                uiBothStep := 1000;

            1000:
                IF Get THEN // Get box job

                    CASE Address_A OF
                        1:
                            DAS_CoreSys.MachineControl.fballocatearea
                                .M_StartStoragePulloutAction(CommandType := E_PullOutConveyorCommandType.SlideB_FeedIn_Ext,
                                                             CV_BackwardTIme := T#0S,
                                                             CV_ForwardTime := T#0S);
                        2:
                            DAS_CoreSys.MachineControl.fballocatearea
                                .M_StartStoragePulloutAction(CommandType := E_PullOutConveyorCommandType.SlideA_FeedIn_Ext,
                                                             CV_BackwardTIme := T#0S,
                                                             CV_ForwardTime := T#0S);
                    END_CASE

                ELSE
                    CASE Address_A OF
                        1:
                            DAS_CoreSys.MachineControl.fballocatearea
                                .M_StartStoragePulloutAction(CommandType := E_PullOutConveyorCommandType.SlideB_FeedOut_Ext,
                                                             CV_BackwardTIme := T#2S,
                                                             CV_ForwardTime := T#0S);

                        2:
                            DAS_CoreSys.MachineControl.fballocatearea
                                .M_StartStoragePulloutAction(CommandType := E_PullOutConveyorCommandType.SlideA_FeedOut_Ext,
                                                             CV_BackwardTIme := T#2S,
                                                             CV_ForwardTime := T#0S);
                    END_CASE

                END_IF

                uiBothStep := 1100;
            1100:
                IF DAS_CoreSys.MachineControl.fballocatearea.fbPulloutCv.Done THEN
                    DAS_CoreSys.MachineControl.fballocatearea.M_StopStoragePulloutAction();
                    BoxReady_1st := TRUE;
                    uiBothStep := 2000;
                END_IF

                IF DAS_CoreSys.MachineControl.fballocatearea.fbPulloutCv.Error THEN
                    DAS_CoreSys.MachineControl.fballocatearea.M_StopStoragePulloutAction();
                    uiResumeStep := 30000;
                    uiBothStep := 1000;
                    _Abort := TRUE;
                    strStatus := 'Feed box timeout';
                END_IF

            2000:
                IF Robot._DI1.Notification THEN
                    uiBothStep := 3000;
                END_IF
            3000:

                IF Get THEN // Get box job

                    CASE Address_B OF
                        1:
                            DAS_CoreSys.MachineControl.fballocatearea
                                .M_StartStoragePulloutAction(CommandType := E_PullOutConveyorCommandType.SlideB_FeedIn_Ext,
                                                             CV_BackwardTIme := T#0S,
                                                             CV_ForwardTime := T#0S);
                        2:
                            DAS_CoreSys.MachineControl.fballocatearea
                                .M_StartStoragePulloutAction(CommandType := E_PullOutConveyorCommandType.SlideA_FeedIn_Ext,
                                                             CV_BackwardTIme := T#0S,
                                                             CV_ForwardTime := T#0S);
                    END_CASE

                ELSE
                    CASE Address_B OF
                        1:
                            DAS_CoreSys.MachineControl.fballocatearea
                                .M_StartStoragePulloutAction(CommandType := E_PullOutConveyorCommandType.SlideB_FeedOut_Ext,
                                                             CV_BackwardTIme := T#2S,
                                                             CV_ForwardTime := T#0S);

                        2:
                            DAS_CoreSys.MachineControl.fballocatearea
                                .M_StartStoragePulloutAction(CommandType := E_PullOutConveyorCommandType.SlideA_FeedOut_Ext,
                                                             CV_BackwardTIme := T#2S,
                                                             CV_ForwardTime := T#0S);
                    END_CASE
                END_IF

                uiBothStep := 3100;
            3100:
                IF DAS_CoreSys.MachineControl.fballocatearea.fbPulloutCv.Done THEN
                    DAS_CoreSys.MachineControl.fballocatearea.M_StopStoragePulloutAction();
                    BoxReady_2nd := TRUE;
                    uiBothStep := 9999;
                END_IF

                IF DAS_CoreSys.MachineControl.fballocatearea.fbPulloutCv.Error THEN
                    DAS_CoreSys.MachineControl.fballocatearea.M_StopStoragePulloutAction();
                    uiResumeStep := 30000;
                    uiBothStep := 3000;
                    _Abort := TRUE;
                    strStatus := 'Feed box timeout';
                END_IF
            9999: //Wait		
        // wait reset
        END_CASE

        // Robot Abs move
        Robot.M_StartRobotAbsMove(GetBox := Get,
                                  UseClampA := UseA,
                                  UseClampB := UseB,
                                  Area := Area,
                                  ClampA_Address := Address_A,
                                  ClampB_Address := Address_B,
                                  BoxReady_1 := BoxReady_1st,
                                  BoxReady_2 := BoxReady_2nd);

        IF Robot._DI1.Done THEN
            tonTimeOut.IN := FALSE;
            uiExecutingStep := 30080;
        END_IF

        tonTimeOut.IN := TRUE;

        IF tonTimeOut.Q = TRUE THEN
            tonTimeOut.IN := FALSE;
            strStatus := 'Reset Robot timeout';
            _Error := TRUE;
        END_IF
    30080: // Check robot command is clear

        Robot.M_ResetRobotAbsMove(UseA, UseB);
        DAS_CoreSys.MachineControl.fballocatearea.M_StopStoragePulloutAction();

        IF NOT Robot._DI1.Done THEN
            tonTimeOut.IN := FALSE;
            uiExecutingStep := 99000; // 
        END_IF

        tonTimeOut.IN := TRUE;

        IF tonTimeOut.Q = TRUE THEN
            strStatus := 'Stop Robot timeout';
            _Error := TRUE;
        END_IF

    99000: // process done
        DAS_CoreSys.MachineControl.fballocatearea.M_ReleasePulloutAccess(ControlAccess := E_RoundBeltControlAccess.FanucRobot);
        Status := 'Process completed';
        _Executed := TRUE;
END_CASE

IF _Executed THEN
    eState := STATE_DONE;
ELSIF _Error THEN
    //	FUN_UniqueErrorCodeGenerator(iErrorID := ErrorID,UinqueErrorCode=>_UniqueErrorCode);
    eState := STATE_ERROR;
ELSIF NOT Execute THEN
    eState := STATE_RESETTING;
END_IF

IF _Abort OR Abort THEN
    //	FUN_UniqueErrorCodeGenerator(iErrorID := ErrorID,UinqueErrorCode=>_UniqueErrorCode);
    eSTATE := STATE_ABORTING;
END_IF
END_METHOD

METHOD  M_STATE_RESETTING
VAR_INPUT
END_VAR
Error := FALSE;
Done := FALSE;
Busy := FALSE;

CASE uiResettingStep OF

    0:
        tonTimeOut.IN := FALSE;
        Robot.M_ResetAllCommand();
        Robot.M_ResetRobotAbsMove(TRUE, TRUE);
        uiResettingStep := 100;
        DAS_CoreSys.MachineControl.fbStorageArea.M_ResetSlides_FeedOut();
    100:

        // DAS_CoreSys.MachineControl.fbStorageArea.M_InactivePulloutConveyorInternCtrl();
        DAS_CoreSys.MachineControl.fbAllocateArea.M_ReleasePulloutAccess(ControlAccess := E_RoundBeltControlAccess.FanucRobot);
        DAS_CoreSys.MachineControl.fbAllocateArea.M_StopStoragePulloutAction();
        uiResettingStep := 9999;
    9999:
        _ResetCompleted := TRUE;
END_CASE

IF _ResetCompleted THEN
    eSTATE := STATE_DORMANT;
END_IF
END_METHOD

END_FUNCTION_BLOCK

// ---- Library/20_MachineUnits/21_StorageArea/Service/FB_RobotRegionMove_RoundBelt.TcPOU
FUNCTION_BLOCK FB_RobotRegionMove_RoundBelt EXTENDS FB_ObjectBase_V2 IMPLEMENTS IBasicElement
VAR_INPUT
    Robot     					: REFERENCE TO FB_FanucRobot_Basic;
	RoundBelt					: REFERENCE TO FB_RoundBeltService;	
   // Command   : ST_WareHouseWithRobotMove_Command;
    Info	  : ST_RobotRegionMove_Info;
	Input : ST_InputTable;
	Stop	  : BOOL;
END_VAR
VAR_OUTPUT
  // Status : ST_WareHouseWithRobotMove_Status;
END_VAR
VAR
	_Abort		: BOOL;
	strStatus	: STRING;
	uiResumeStep : UINT;
	
	Area	: E_RobotArea :=E_RobotArea.RoundBelt;
	UseA 	: BOOL;
	UseB	: BOOL;
	
	Get 	:BOOL;
	tonTimeOut	:TON;
	tonCheckRoundBeltDelay	:TON;
	_UniqueErrorCode :STRING;
	PreviousStrStatus : STRING;
	PreviousErrorCode : STRING;
END_VAR

SUPER^.A10_StateControl();
A00_BasicUnits();

ACTION A00_BasicUnits:
tonTimeOut(PT:=T#60S);
tonCheckRoundBeltDelay(PT:=T#2S);
ErrorID:=2220;
END_ACTION

METHOD M_CheckCommand : BOOL // True : Command is useful
VAR_INPUT
END_VAR
VAR
	
END_VAR
// Check command paremeter is correct
	
THIS^.Get :=Info.Get;
UseA := Info.UseA;
UseB := Info.UseB;
	//Normal command : RoundBelt
		IF Info.UseA AND (Info.A_Position<1 OR  Info.A_Position>3) THEN
			strStatus:='Wrong command ,Position A Not allowed';
			M_CheckCommand:=FALSE;
			RETURN;			
		END_IF
		
	
	//Normal command : RoundBelt
		IF Info.UseB AND(Info.B_Position<1 OR  Info.B_Position>3) THEN
			strStatus:='Wrong command ,Position B Not allowed';
			M_CheckCommand:=FALSE;
			RETURN;				
		END_IF
		
	

M_CheckCommand:=TRUE;
END_METHOD

METHOD M_CheckUnitsNotBusy : BOOL
VAR_INPUT
END_VAR
M_CheckUnitsNotBusy := true;
END_METHOD

METHOD M_CheckUnitsReady : BOOL
VAR_INPUT
END_VAR
M_CheckUnitsReady := true;
END_METHOD

METHOD  M_STATE_ABORTED
VAR_INPUT
END_VAR
ERROR :=TRUE;
Busy    := FALSE;
Aborted := TRUE;
Status := strStatus;
UniqueErrorCode:=_UniqueErrorCode;
IF NOT Execute THEN
	eSTATE:=STATE_RESETTING;
END_IF

IF Execute AND Reset THEN
	PreviousStrStatus := strStatus;
	PreviousErrorCode := _UniqueErrorCode;
	uiExecutingStep :=uiResumeStep;
	eSTATE:=STATE_EXECUTING;
END_IF
END_METHOD

METHOD  M_STATE_ABORTING
VAR_INPUT
END_VAR
CASE uiAbortingStep OF
	0 :
		uiAbortingStep:=9999;
		tonTimeOut.IN :=FALSE;
		_Abort :=FALSE;
		IF strStatus = PreviousStrStatus THEN
			_UniqueErrorCode :=PreviousErrorCode;
		END_IF
	9999:	_AbortCompleted:=TRUE;
END_CASE

IF _AbortCompleted THEN	
	eSTATE :=STATE_ABORTED;
END_IF
END_METHOD

METHOD  M_STATE_DONE
VAR_INPUT
END_VAR
Busy := FALSE;
Done := TRUE;
IF NOT Execute THEN
    eState := STATE_RESETTING;
END_IF
END_METHOD

METHOD  M_STATE_DORMANT
VAR_INPUT
END_VAR
// Clear FB output
Busy            := FALSE;
Done            := FALSE;
Aborted         := FALSE;
Error           := FALSE;
ErrorID         := 0;
Status          := '';
_ResetCompleted := FALSE;
_Error          := FALSE;
_Executed       := FALSE;

tonTimeOut.IN:=tonCheckRoundBeltDelay.IN:= FALSE;
strStatus :='No Error';
uiExecutingStep :=uiResettingStep :=uiResumeStep :=0;
PreviousStrStatus			 :='';
PreviousErrorCode			 :='';

// Wait Execute command
IF Execute THEN
    eState := STATE_EXECUTING;
END_IF
END_METHOD

METHOD  M_STATE_ERROR
VAR_INPUT
END_VAR
ERROR   :=TRUE;
Busy	:=FALSE;
Status := strStatus;
UniqueErrorCode:=_UniqueErrorCode;
IF NOT Execute THEN	
eSTATE:=STATE_RESETTING;
END_IF
END_METHOD

METHOD  M_STATE_EXECUTING
VAR_INPUT
END_VAR
VAR_INST
	BoxReady_1st : BOOL;
	BoxReady_2nd : BOOL;
    uiBothStep : UINT;
    uiSingleClampStep : UINT;	
	Address_A : INT;
	Address_B : INT;
	A1Used	 : BOOL;
	A2Used	 : BOOL;
END_VAR
VAR
	
	
END_VAR
//20250418 note: current behavior : wait round belt finish rotating then check if box is ready , everything ready then call Robot start move
//				 Todo : consider if better call robot start move to waiting position and check box at same moment , Albert 

// Set Busy active edit by johnson
Busy := TRUE;
IF THIS^.Stop THEN // Pending the timeout when Stop signal occur
	tonTimeout.IN :=FALSE;
END_IF
// Service Process
CASE uiExecutingStep OF
	0:
        // Clear variable      
        uiBothStep := 0;
		uiSingleClampStep :=0;
		BoxReady_1st := 0;
		BoxReady_2nd := 0;
		tonTimeOut.IN:=FALSE;
		tonCheckRoundBeltDelay.IN :=FALSE;
        // Check command
        IF M_CheckCommand() THEN
            uiExecutingStep := 10;
		ELSE
			_Error:=TRUE;
        END_IF
    10:
        // Start process, check units first
        IF M_CheckUnitsReady() THEN
            uiExecutingStep := 20;
        END_IF
    20:
        // CHeck units not busy state
        IF M_CheckUnitsNotBusy() THEN
            uiExecutingStep := 1000;
        END_IF
   
	1000:   
			// Read   coordinate
			 Area := THIS^.Area;
 			 Address_A := LREAL_TO_INT(Info.A_Position);
			 Address_B := LREAL_TO_INT(Info.B_Position);
			 uiExecutingStep := 1100; 		
			 
	1100:	
			// Check clamp userage	 
			IF UseA AND NOT UseB THEN
				//Only clampA
				uiExecutingStep := 10000;
			ELSIF NOT UseA AND UseB THEN
				//Only ClampB 
				uiExecutingStep := 20000;
			ELSIF UseA AND UseB THEN
				//Both Clamps
				uiExecutingStep := 30000;		
			END_IF
       
    10000: // Only ClampA 
        IF NOT Robot._DI1.Done THEN
			// Delay to make sure round belt is starting/finish rotating
			IF NOT RoundBelt.xBusy AND NOT RoundBelt.xError THEN
				tonCheckRoundBeltDelay.IN:=TRUE;
			ELSE
				tonCheckRoundBeltDelay.IN:=FALSE;	
			END_IF
		
		
		CASE uiSingleClampStep OF
		0:
			CASE Address_A OF						
						1: A1Used := TRUE;
						2: A2Used := TRUE;
			END_CASE
			
			IF tonCheckRoundBeltDelay.Q THEN
				IF Get THEN  // Picking job , check box is ready
					IF A1Used AND Input.bRoundBelt_ChangeZoneA2Detect_Sensor =FALSE	THEN
						_Error:=TRUE	;
						strStatus :='No Box on A1';
					END_IF				
					IF A2Used AND Input.bRoundBelt_ChangeZoneA3Detect_Sensor =FALSE	THEN
						_Error:=TRUE	;
						strStatus :='No Box on A2';
					END_IF	
				ELSE		//Place job , check no box 
					IF A1Used AND Input.bRoundBelt_ChangeZoneA2Detect_Sensor =TRUE	THEN
						_Error:=TRUE	;
						strStatus :='Box on A1';
					END_IF				
					IF A2Used AND Input.bRoundBelt_ChangeZoneA3Detect_Sensor =TRUE	THEN
						_Error:=TRUE	;
						strStatus :='Box on A2';
					END_IF				
				END_IF
				 uiSingleClampStep:=100;  
			END_IF
	  
		  100 :  
		  		IF get THEN
					BoxReady_1st := (A1Used AND Input.bRoundBelt_ChangeZoneA2Detect_Sensor) OR
		  						 (A2Used AND Input.bRoundBelt_ChangeZoneA3Detect_Sensor);
				ELSE
					BoxReady_1st := (A1Used AND NOT Input.bRoundBelt_ChangeZoneA2Detect_Sensor) OR
		  						 (A2Used AND NOT Input.bRoundBelt_ChangeZoneA3Detect_Sensor);
				END_IF		
				IF BoxReady_1st THEN
					uiSingleClampStep:=9999;  
				END_IF			 
								 
		  9999:// 
	
		END_CASE				          		 
				  // Robot Abs move
           		 Robot.M_StartRobotAbsMove(GetBox:=Get,
											UseClampA:=UseA,
											UseClampB:=UseB,
											Area:=Area,
											ClampA_Address:=Address_A,
											ClampB_Address:=Address_B,
											BoxReady_1:=BoxReady_1st,
											BoxReady_2:=BoxReady_2nd);				  
		
        ELSE
			tonTimeOut.IN:=FALSE;
            uiExecutingStep := 10080;
        END_IF
		tonTimeOut.IN:=TRUE;
		IF tonTimeOut.Q=TRUE THEN
			tonTimeOut.IN:=FALSE;
			strStatus :='Reset Robot timeout';
			_Error:=TRUE;
		END_IF	
    10080:
        Robot.M_ResetRobotAbsMove(UseA,UseB); // Clear command and go to place box
		tonTimeOut.IN:=TRUE;
        IF NOT Robot._DI1.Done THEN
			tonTimeOut.IN:=FALSE;
            uiExecutingStep := 99000; 
        END_IF
    	IF tonTimeOut.Q=TRUE THEN
			strStatus :='Reset Robot timeout';
			_Error:=TRUE;
		END_IF	
    
   20000: // Only ClampB
        IF NOT Robot._DI1.Done THEN
           IF NOT RoundBelt.xBusy AND NOT RoundBelt.xError THEN
				tonCheckRoundBeltDelay.IN:=TRUE;
			ELSE
				tonCheckRoundBeltDelay.IN:=FALSE;	
			END_IF
		
		
		CASE uiSingleClampStep OF
		0:
			CASE Address_B OF						
						1: A1Used := TRUE;
						2: A2Used := TRUE;
			END_CASE
			
			IF tonCheckRoundBeltDelay.Q THEN
				IF Get THEN  // Picking job , check box is ready
					IF A1Used AND Input.bRoundBelt_ChangeZoneA2Detect_Sensor =FALSE	THEN
						_Error:=TRUE	;
						strStatus :='No Box on A1';
					END_IF				
					IF A2Used AND Input.bRoundBelt_ChangeZoneA3Detect_Sensor =FALSE	THEN
						_Error:=TRUE	;
						strStatus :='No Box on A2';
					END_IF	
				ELSE		//Place job , check no box 
					IF A1Used AND Input.bRoundBelt_ChangeZoneA2Detect_Sensor =TRUE	THEN
						_Error:=TRUE	;
						strStatus :='Box on A1';
					END_IF				
					IF A2Used AND Input.bRoundBelt_ChangeZoneA3Detect_Sensor =TRUE	THEN
						_Error:=TRUE	;
						strStatus :='Box on A2';
					END_IF				
				END_IF
				 uiSingleClampStep:=100;  
			END_IF
	  
		  100 :  
		  		IF get THEN
					BoxReady_2nd := (A1Used AND Input.bRoundBelt_ChangeZoneA2Detect_Sensor) OR
		  						 (A2Used AND Input.bRoundBelt_ChangeZoneA3Detect_Sensor);
				ELSE
					BoxReady_2nd := (A1Used AND NOT Input.bRoundBelt_ChangeZoneA2Detect_Sensor) OR
		  						 (A2Used AND NOT Input.bRoundBelt_ChangeZoneA3Detect_Sensor);
				END_IF		
				IF BoxReady_2nd THEN
					uiSingleClampStep:=9999;  
				END_IF			 
								 
		  9999:// 
	
		END_CASE				          		 
					  // Robot Abs move
           		 Robot.M_StartRobotAbsMove( GetBox:=Get,
											UseClampA:=UseA,
											UseClampB:=UseB,
											Area:=Area,
											ClampA_Address:=Address_A,
											ClampB_Address:=Address_B,
											BoxReady_1:=BoxReady_1st,
											BoxReady_2:=BoxReady_2nd);		  
		
        ELSE
			tonTimeOut.IN:=FALSE;
            uiExecutingStep := 20080;
        END_IF	
		tonTimeOut.IN:=TRUE;
		IF tonTimeOut.Q=TRUE THEN
			tonTimeOut.IN:=FALSE;
			strStatus :='Reset Robot timeout';
			_Error:=TRUE;
		END_IF				          		 
			
       
		
    20080:
       Robot.M_ResetRobotAbsMove(UseA,UseB);; // Clear command 

        IF NOT Robot._DI1.Done THEN
            uiExecutingStep := 99000; 
        END_IF
		tonTimeOut.IN:=TRUE;
		IF tonTimeOut.Q=TRUE THEN
			strStatus :='Reset Robot timeout';
			_Error:=TRUE;
		END_IF	
    30000: // Both Clamps
        	
			IF NOT RoundBelt.xBusy AND NOT RoundBelt.xError THEN
				tonCheckRoundBeltDelay.IN:=TRUE;
			ELSE
				tonCheckRoundBeltDelay.IN:=FALSE;	
			END_IF
		
		  CASE uiBothStep OF
           		0://	
					BoxReady_1st := FALSE;
					BoxReady_2nd := FALSE;
					
					IF tonCheckRoundBeltDelay.Q THEN
						uiBothStep:=100;	
					END_IF
				100:
					IF Get THEN  // Picking job , check box is ready
						IF  Input.bRoundBelt_ChangeZoneA2Detect_Sensor =FALSE	THEN
							_Error:=TRUE	;
							strStatus :='No Box on A1';
						END_IF				
						IF  Input.bRoundBelt_ChangeZoneA3Detect_Sensor =FALSE	THEN
							_Error:=TRUE	;
							strStatus :='No Box on A2';
						END_IF	
					ELSE		//Place job , check no box 
						IF  Input.bRoundBelt_ChangeZoneA2Detect_Sensor =TRUE	THEN
							_Error:=TRUE	;
							strStatus :='Box on A1';
						END_IF				
						IF  Input.bRoundBelt_ChangeZoneA3Detect_Sensor =TRUE	THEN
							_Error:=TRUE	;
							strStatus :='Box on A2';
						END_IF				
					END_IF
					IF NOT _Error THEN
						uiBothStep:=1000;
					END_IF
				1000:	
						
						BoxReady_1st :=TRUE;
						uiBothStep:=2000;
					
						
				2000:					
						IF Robot._DI1.Notification THEN
							uiBothStep:=3000;
						END_IF
				3000:	
						 BoxReady_2nd :=TRUE;						 
					     uiBothStep:=9999;
				
				9999: //Wait		
        // wait reset
        END_CASE

       	  // Robot Abs move
           		 Robot.M_StartRobotAbsMove( GetBox:=Get,
											UseClampA:=UseA,
											UseClampB:=UseB,
											Area:=Area,
											ClampA_Address:=Address_A,
											ClampB_Address:=Address_B,
											BoxReady_1:=BoxReady_1st,
											BoxReady_2:=BoxReady_2nd);	
		
		
        IF Robot._DI1.Done THEN
			tonTimeOut.IN:=FALSE;
            uiExecutingStep := 30080;
        END_IF
		tonTimeOut.IN:=TRUE;
		IF tonTimeOut.Q=TRUE THEN
			tonTimeOut.IN:=FALSE;
			strStatus :='Reset Robot timeout';
			_Error:=TRUE;
		END_IF	
		
    30080: // Check robot command is clear
        
        Robot.M_ResetRobotAbsMove(UseA,UseB);

        IF NOT Robot._DI1.Done THEN
			tonTimeOut.IN:=FALSE;
            uiExecutingStep := 99000; // go to place step
        END_IF    
   		tonTimeOut.IN:=TRUE;
		IF tonTimeOut.Q=TRUE THEN
			strStatus :='Stop Robot timeout';
			_Error:=TRUE;
		END_IF	
   
    99000:
			IF Get THEN  // Picking job , check box putted
				IF A1Used AND Input.bRoundBelt_ChangeZoneA2Detect_Sensor =TRUE	THEN
					_Error:=TRUE	;
					strStatus :='Box still on A1';
				END_IF				
				IF A2Used AND Input.bRoundBelt_ChangeZoneA3Detect_Sensor =TRUE	THEN
					_Error:=TRUE	;
					strStatus :='No still on A2';
				END_IF	
			ELSE		//Place job , check no box 
				IF A1Used AND Input.bRoundBelt_ChangeZoneA2Detect_Sensor =FALSE	THEN
					_Error:=TRUE	;
					strStatus :='No Box on A1';
				END_IF				
				IF A2Used AND Input.bRoundBelt_ChangeZoneA3Detect_Sensor =FALSE	THEN
					_Error:=TRUE	;
					strStatus :='No Box on A2';
				END_IF	
			
			END_IF
			IF NOT _Error THEN
			 	uiExecutingStep := 99100;
			 END_IF
	99100: // process done
                Status    := 'Process completed';
        	_Executed := TRUE;
END_CASE
IF _Executed THEN
    eState := STATE_DONE;
ELSIF _Error THEN
//	FUN_UniqueErrorCodeGenerator(iErrorID := ErrorID,UinqueErrorCode=>_UniqueErrorCode);
    eState := STATE_ERROR;
ELSIF NOT Execute THEN
    eState := STATE_RESETTING;
END_IF
IF _Abort OR Abort THEN
//	FUN_UniqueErrorCodeGenerator(iErrorID := ErrorID,UinqueErrorCode=>_UniqueErrorCode);
	eSTATE:=STATE_ABORTING;
END_IF
END_METHOD

METHOD  M_STATE_RESETTING
VAR_INPUT
END_VAR
Error :=FALSE;
Done :=FALSE;
Busy := FALSE;


CASE uiResettingStep OF
	
	0:
		tonTimeOut.IN:=FALSE;
		Robot.M_ResetAllCommand();
		Robot.M_ResetRobotAbsMove(TRUE,TRUE);
		uiResettingStep:=100;
		
	100:
	
		uiResettingStep:=9999;
	9999:
		_ResetCompleted:=TRUE;
END_CASE
IF _ResetCompleted THEN
	eSTATE:=STATE_DORMANT;
END_IF
END_METHOD

END_FUNCTION_BLOCK

// ---- Library/20_MachineUnits/21_StorageArea/Service/FB_RobotAbsMove.TcPOU
FUNCTION_BLOCK FB_RobotAbsMove EXTENDS FB_ObjectBase_V2 IMPLEMENTS IBasicElement
VAR_INPUT
    Robot         : REFERENCE TO FB_FanucRobot_Basic;
    LowerConveyor : REFERENCE TO FB_Motor;
    // Command   : ST_WareHouseWithRobotMove_Command;
    Info : st_AutoSixAxisAbsMoveParameter;
	Input :ST_InputTable;
    Stop : BOOL;
END_VAR
VAR_OUTPUT
    // Status : ST_WareHouseWithRobotMove_Status;
END_VAR
VAR
    _Abort       : BOOL;
    strStatus    : STRING;
    uiResumeStep : UINT;

    Area : E_RobotArea;
    UseA : BOOL;
    UseB : BOOL;

    Get                         : BOOL;
    tonTimeOut                  : TON;
	TON_DelayLowerCV			: TON;
    _UniqueErrorCode            : STRING;
    FirstSensorOfLowerConveyor  : BOOL;
    SecondSensorOfLowerConveyor : BOOL;

END_VAR

SUPER^.A10_StateControl();
A00_BasicUnits();
FirstSensorOfLowerConveyor := Input.bLowCV_BoxArrived_Sensor;
SecondSensorOfLowerConveyor := Input.bLowCV_2ndBoxGap_Sensor;

ACTION A00_BasicUnits:
tonTimeOut(PT:=T#60S);
TON_DelayLowerCV(PT:=T#1S);
ErrorID :=2200;
END_ACTION

METHOD M_CheckCommand : BOOL // True : Command is useful
VAR_INPUT
END_VAR
VAR
	
END_VAR
// Check command paremeter is correct


IF Info.A_Get <> Info.B_Get THEN
	strStatus:='Wrong command ,GetA not match to GetB';
	M_CheckCommand:=FALSE;
	RETURN;
ELSE		
	THIS^.Get :=Info.A_Get;
END_IF

IF Info.A_Area<> Info.B_Area THEN
	IF NOT(Info.A_Area=99 OR Info.B_Area=99) THEN
	strStatus:='Wrong command ,Area A not match to Area B';
	M_CheckCommand:=FALSE;
	RETURN;
END_IF
END_IF

IF Info.A_Area = 99 AND Info.B_Area = 99 THEN
	strStatus:='Wrong command ,Both Area are 99';
	M_CheckCommand:=FALSE;
	RETURN;
END_IF

CASE LREAL_TO_INT(Info.A_Area) OF
	1 : //Normal command : RoundBelt
		IF Info.A_Position<1 OR  Info.A_Position>3 THEN
			strStatus:='Wrong command ,Position A Not allow';
			M_CheckCommand:=FALSE;
			RETURN;	
		ELSE
			Area := E_RobotArea.RoundBelt;
			UseA :=TRUE	;	
		END_IF
		
	2:	//Buffer area
		IF Info.A_Position<1 OR  Info.A_Position>40 THEN
			strStatus:='Wrong command ,Position A Not allow';
			M_CheckCommand:=FALSE;
			RETURN;	
		ELSE
			Area := E_RobotArea.BufferArea;
			UseA :=TRUE	;	
		END_IF
	3: //Allocated/Empty conveyor
		IF Info.A_Position<1 OR  Info.A_Position>2 THEN
			strStatus:='Wrong command ,Position A Not allow';
			M_CheckCommand:=FALSE;
			RETURN;	
		ELSE
			Area := E_RobotArea.TransmitCV;
			UseA :=TRUE	;	
		END_IF
	5: //FeedIn/Out conveyor
		IF Info.A_Position<1 OR  Info.A_Position>3 THEN
			strStatus:='Wrong command ,Position A Not allow';
			M_CheckCommand:=FALSE;
			RETURN;	
		ELSIF Info.A_Position=3 AND Get THEN
			strStatus:='Wrong command ,Can Not Get box from FeedOut conveyor ';
			M_CheckCommand:=FALSE;
			RETURN;	
		ELSE
			Area := E_RobotArea.InOutConveyor;
			UseA :=TRUE	;	
		END_IF
	7: // PullOut conveyor
		IF Info.A_Position<1 OR  Info.A_Position>2 THEN
			strStatus:='Wrong command ,Position A Not allow';
			M_CheckCommand:=FALSE;
			RETURN;	
		ELSE
			Area := E_RobotArea.PullOutConveyor;
			UseA :=TRUE	;	
		END_IF
	
	99: //ClampA not use
		UseA :=FALSE;
	
	ELSE //Wrong command
		strStatus:='Wrong command ,Area_A not allow ';
		M_CheckCommand:=FALSE;
		RETURN;

END_CASE

CASE LREAL_TO_INT(Info.B_Area) OF
	1 : //Normal command : RoundBelt
		IF Info.B_Position<1 OR  Info.B_Position>3 THEN
			strStatus:='Wrong command ,Position B Not allow';
			M_CheckCommand:=FALSE;
			RETURN;	
		ELSE
			Area := E_RobotArea.RoundBelt;
			UseB :=TRUE	;	
		END_IF
		
	2:	
		IF Info.B_Position<1 OR  Info.B_Position>40 THEN
			strStatus:='Wrong command ,Position B Not allow';
			M_CheckCommand:=FALSE;
			RETURN;	
		ELSE
			Area := E_RobotArea.BufferArea;
			UseB :=TRUE	;	
		END_IF
	3:
		IF Info.B_Position<1 OR  Info.B_Position>2 THEN
			strStatus:='Wrong command ,Position B Not allow';
			M_CheckCommand:=FALSE;
			RETURN;	
		ELSE
			Area := E_RobotArea.TransmitCV;
			UseB :=TRUE	;	
		END_IF
	5:
		IF Info.B_Position<1 OR  Info.B_Position>3 THEN
			strStatus:='Wrong command ,Position B Not allow';
			M_CheckCommand:=FALSE;
			RETURN;	
		ELSE
			Area := E_RobotArea.InOutConveyor;
			UseB :=TRUE	;	
		END_IF
	7:
		IF Info.B_Position<1 OR  Info.B_Position>2 THEN
			strStatus:='Wrong command ,Position B Not allow';
			M_CheckCommand:=FALSE;
			RETURN;	
		ELSIF Info.B_Position=3 AND Get THEN
			strStatus:='Wrong command ,Can Not Get box from FeedOut conveyor ';
			M_CheckCommand:=FALSE;
			RETURN;	
		ELSE
			Area := E_RobotArea.PullOutConveyor;
			UseB :=TRUE	;	
		END_IF
	
	99: //ClampA not use
		UseB :=FALSE;
	
	ELSE //Wrong command
		strStatus:='Wrong command ,Area_B not allow ';
		M_CheckCommand:=FALSE;
		RETURN;

END_CASE


M_CheckCommand:=TRUE;
END_METHOD

METHOD M_CheckUnitsNotBusy : BOOL
VAR_INPUT
END_VAR
M_CheckUnitsNotBusy := true;
END_METHOD

METHOD M_CheckUnitsReady : BOOL
VAR_INPUT
END_VAR
M_CheckUnitsReady := true;
END_METHOD

METHOD  M_STATE_ABORTED
VAR_INPUT
END_VAR
ERROR :=TRUE;
Busy    := FALSE;
Aborted := TRUE;
Status := strStatus;
UniqueErrorCode:=_UniqueErrorCode;
IF NOT Execute THEN
	eSTATE:=STATE_RESETTING;
END_IF

IF Execute AND Reset THEN
	uiExecutingStep :=uiResumeStep;
	eSTATE:=STATE_EXECUTING;
END_IF
END_METHOD

METHOD  M_STATE_ABORTING
VAR_INPUT
END_VAR
CASE uiAbortingStep OF
	0 :
		uiAbortingStep:=9999;
	
	9999:	_AbortCompleted:=TRUE;
END_CASE

IF _AbortCompleted THEN	
	eSTATE :=STATE_ABORTED;
END_IF
END_METHOD

METHOD  M_STATE_DONE
VAR_INPUT
END_VAR
Busy := FALSE;
Done := TRUE;
IF NOT Execute THEN
    eState := STATE_RESETTING;
END_IF
END_METHOD

METHOD  M_STATE_DORMANT
VAR_INPUT
END_VAR
// Clear FB output
Busy            := FALSE;
Done            := FALSE;
Aborted         := FALSE;
Error           := FALSE;
ErrorID         := 0;
Status          := '';
_ResetCompleted := FALSE;
_Error          := FALSE;
_Executed       := FALSE;

tonTimeOut.IN:=FALSE;
TON_DelayLowerCV.IN := false;
strStatus :='No Error';
uiExecutingStep :=uiResettingStep :=uiResumeStep :=0;


// Wait Execute command
IF Execute THEN
    eState := STATE_EXECUTING;
END_IF
END_METHOD

METHOD  M_STATE_ERROR
VAR_INPUT
END_VAR
ERROR   :=TRUE;
Busy	:=FALSE;
Status := strStatus;
UniqueErrorCode:=_UniqueErrorCode;
ErrorID :=2200;
IF NOT Execute THEN	
eSTATE:=STATE_RESETTING;
END_IF
END_METHOD

METHOD  M_STATE_EXECUTING
VAR_INPUT
END_VAR
VAR_INST
    ActionMode       : E_ReloadRoundBoxAction;
	BoxReady_1st : BOOL;
	BoxReady_2nd : BOOL;
    CarrierReady_1st : BOOL;
    CarrierReady_2nd : BOOL;
    uiBothStep : UINT;
    uiSingleClampStep : UINT;	
	Area : E_RobotArea;
	Address_A : INT;
	Address_B : INT;
END_VAR
VAR
	WareHouse: INT;
END_VAR
// Set Busy active edit by johnson
Busy := TRUE;
IF THIS^.Stop THEN // Pending the timeout when Stop signal occur
	tonTimeout.IN :=FALSE;
END_IF
// Service Process
CASE uiExecutingStep OF
	0:
        // Clear variable
        ActionMode       := E_ReloadRoundBoxAction.Undefined;
        CarrierReady_1st := FALSE;
        CarrierReady_2nd := FALSE;
        uiBothStep := 0;
		uiSingleClampStep :=0;
		BoxReady_1st := 0;
		BoxReady_2nd := 0;
		tonTimeOut.IN:=FALSE;
        // Check command
        IF M_CheckCommand() THEN
            uiExecutingStep := 10;
		ELSE
			_Error:=TRUE;
        END_IF
    10:
        // Start process, check units first
        IF M_CheckUnitsReady() THEN
            uiExecutingStep := 20;
        END_IF
    20:
        // CHeck units not busy state
        IF M_CheckUnitsNotBusy() THEN
            uiExecutingStep := 1000;
        END_IF
   
	1000:   
			// Read   coordinate
			 Area := THIS^.Area;
 			 Address_A := LREAL_TO_INT(Info.A_Position);
			 Address_B := LREAL_TO_INT(Info.B_Position);
			 
			IF UseA AND NOT UseB THEN
				//Only clampA
				uiExecutingStep := 10000;
			ELSIF NOT UseA AND UseB THEN
				//Only ClampB 
				uiExecutingStep := 20000;
			ELSIF UseA AND UseB THEN
				//Both Clamps
				uiExecutingStep := 30000;		
			END_IF
       
    10000: // Only ClampA 
        IF NOT Robot._DI1.Done THEN
            
            
			CASE uiSingleClampStep OF
				
				0://
					IF Area= E_RobotArea.InOutConveyor AND Address_A=3 THEN
						uiSingleClampStep:=100;// Need to control feedout conveyor 
					ELSE
						uiSingleClampStep:=1000;	
					END_IF
				100:	//check the box is full 
					IF Input.bLowCV_Block2Detect_Sensor THEN 
						_Error := TRUE;
						strStatus :='LowerCV the box behind is full, please remove it';
					ELSE 
						uiSingleClampStep := 150;
					END_IF
				
				150:	//check the box not no the  sensor 
					IF  FirstSensorOfLowerConveyor OR  (NOT SecondSensorOfLowerConveyor) THEN
						LowerConveyor.M_MoveBackward();
						tonTimeOut.IN:=FALSE;;
						uiSingleClampStep:=200;
					ELSE 
						uiSingleClampStep := 1000;
					END_IF
					tonTimeOut.IN:=TRUE;
					IF tonTimeOut.Q=TRUE THEN
						strStatus :='Empty Conveyor timeout';
						_Error:=TRUE;
					END_IF
				200:
//					TON_DelayLowerCV.IN := TRUE;
//					IF TON_DelayLowerCV.Q THEN
//					LowerConveyor.M_MotorStop();
//					uiSingleClampStep:=300;
//					END_IF 
					IF Input.bLowCV_Block2Detect_Sensor THEN
						TON_DelayLowerCV.IN := TRUE;
					END_IF
					IF TON_DelayLowerCV.Q THEN
						LowerConveyor.M_MotorStop();
						uiSingleClampStep := 300;
					END_IF
									
				300:
					TON_DelayLowerCV.IN :=FALSE;
					IF 	LowerConveyor.InStopped THEN
						tonTimeOut.IN:=FALSE;
						uiSingleClampStep:=1000;
					END_IF
					tonTimeOut.IN:=TRUE;
					IF tonTimeOut.Q=TRUE THEN
						strStatus :='Stop Conveyor timeout';
						_Error:=TRUE;
					END_IF	
				1000:
						BoxReady_1st:=TRUE;
						uiSingleClampStep:=9999;
				9999: //Wait	
			END_CASE
			          		 
				  // Robot Abs move
           		 Robot.M_StartRobotAbsMove(GetBox:=Get,
											UseClampA:=UseA,
											UseClampB:=UseB,
											Area:=Area,
											ClampA_Address:=Address_A,
											ClampB_Address:=Address_B,
											BoxReady_1:=BoxReady_1st,
											BoxReady_2:=BoxReady_2nd);				  
		
        ELSE
            uiExecutingStep := 10080;
        END_IF
		
    10080:
        Robot.M_ResetRobotAbsMove(UseA,UseB); // Clear command and go to place box
		tonTimeOut.IN:=TRUE;
        IF NOT Robot._DI1.Done THEN
			tonTimeOut.IN:=FALSE;
            uiExecutingStep := 40000; 
        END_IF
    	IF tonTimeOut.Q=TRUE THEN
			strStatus :='Reset Robot timeout';
			_Error:=TRUE;
		END_IF
		
    
   20000: // Only ClampB
        IF NOT Robot._DI1.Done THEN
            			
			CASE uiSingleClampStep OF
				
				0://
					IF Area= E_RobotArea.InOutConveyor AND Address_B=3 THEN
						uiSingleClampStep:=100;// Need to control feedout conveyor 
					ELSE
						uiSingleClampStep:=1000;	
					END_IF
					
				100:	//check the box is full 
					IF Input.bLowCV_Block2Detect_Sensor THEN 
						_Error := TRUE;
						strStatus :='LowerCV the box behind is full, please remove it';
					ELSE 
						uiSingleClampStep := 150;
					END_IF
				
				150:	//check the box not no the  sensor 
					IF  FirstSensorOfLowerConveyor OR  (NOT SecondSensorOfLowerConveyor) THEN
						LowerConveyor.M_MoveBackward();
						tonTimeOut.IN:=FALSE;;
						uiSingleClampStep:=200;
					ELSE
						uiSingleClampStep := 1000;
					END_IF
					tonTimeOut.IN:=TRUE;
					IF tonTimeOut.Q=TRUE THEN
						strStatus :='Empty Conveyor timeout';
						_Error:=TRUE;
					END_IF
				200:
//					TON_DelayLowerCV.IN := TRUE;
//					IF TON_DelayLowerCV.Q THEN
//					LowerConveyor.M_MotorStop();
//					uiSingleClampStep:=300;
//					END_IF 
					IF Input.bLowCV_Block2Detect_Sensor THEN
						TON_DelayLowerCV.IN := TRUE;
					END_IF
					IF TON_DelayLowerCV.Q THEN
						LowerConveyor.M_MotorStop();
						uiSingleClampStep := 300;
					END_IF
									
				300:
					TON_DelayLowerCV.IN :=FALSE;
					IF 	LowerConveyor.InStopped THEN
						tonTimeOut.IN:=FALSE;
						uiSingleClampStep:=1000;
					END_IF
					tonTimeOut.IN:=TRUE;
					IF tonTimeOut.Q=TRUE THEN
						strStatus :='Stop Conveyor timeout';
						_Error:=TRUE;
					END_IF	
				1000:
						BoxReady_2nd:=TRUE;
						uiSingleClampStep:=9999;
				9999: //Wait			
			END_CASE
			          		 
				  // Robot Abs move
           		 Robot.M_StartRobotAbsMove( GetBox:=Get,
											UseClampA:=UseA,
											UseClampB:=UseB,
											Area:=Area,
											ClampA_Address:=Address_A,
											ClampB_Address:=Address_B,
											BoxReady_1:=BoxReady_1st,
											BoxReady_2:=BoxReady_2nd);	
        ELSE
            uiExecutingStep := 20080;
        END_IF
		
    20080:
       Robot.M_ResetRobotAbsMove(UseA,UseB);; // Clear command 

        IF NOT Robot._DI1.Done THEN
            uiExecutingStep := 40000; 
        END_IF
		tonTimeOut.IN:=TRUE;
		IF tonTimeOut.Q=TRUE THEN
			strStatus :='Reset Robot timeout';
			_Error:=TRUE;
		END_IF	
    30000: // Both Clamps
        		
		
		  CASE uiBothStep OF
           		0://	
					BoxReady_1st := FALSE;
					BoxReady_2nd := FALSE;
					IF Area= E_RobotArea.InOutConveyor AND Address_A=3 THEN
						uiBothStep:=100;// Need to control feedout conveyor 
					ELSE
						uiBothStep:=1000;	
					END_IF
					
				100:	//check the box is full 
					IF Input.bLowCV_Block2Detect_Sensor THEN 
						_Error := TRUE;
						strStatus :='LowerCV the box behind is full, please remove it';
					ELSE 
						uiBothStep := 200;
					END_IF
				
				200:	//check the box not no the  sensor 
					IF  FirstSensorOfLowerConveyor OR  (NOT SecondSensorOfLowerConveyor) THEN
						LowerConveyor.M_MoveBackward();
						tonTimeOut.IN:=FALSE;;
						uiBothStep:=300;
					ELSE
						uiBothStep := 1000;
					END_IF
					tonTimeOut.IN:=TRUE;
					IF tonTimeOut.Q=TRUE THEN
						strStatus :='Empty Conveyor timeout';
						_Error:=TRUE;
					END_IF
				300:
					IF Input.bLowCV_Block2Detect_Sensor THEN
						TON_DelayLowerCV.IN := TRUE;
					END_IF
					IF TON_DelayLowerCV.Q THEN
						LowerConveyor.M_MotorStop();
						uiBothStep := 400;
					END_IF
								
				400:
					TON_DelayLowerCV.IN :=FALSE;
					IF 	LowerConveyor.InStopped THEN
						tonTimeOut.IN:=FALSE;
						uiBothStep:=1000;
					END_IF
					tonTimeOut.IN:=TRUE;
					IF tonTimeOut.Q=TRUE THEN
						strStatus :='Stop Robot timeout';
						_Error:=TRUE;
					END_IF		
				1000:
						BoxReady_1st:=TRUE;
						uiBothStep:=2000;
						
				2000:
						IF Robot._DI1.Notification THEN
							uiBothStep:=3000;
						END_IF
				3000:
					
					IF Area= E_RobotArea.InOutConveyor AND Address_B=3 THEN
						uiBothStep:=3100;// Need to control feedout conveyor 
					ELSE
						uiBothStep:=9000;	
					END_IF
					
				3100:
					IF Input.bLowCV_Block2Detect_Sensor THEN 
						_Error := TRUE;
						strStatus :='LowerCV the box behind is full, please remove it';
					ELSE 
						uiBothStep := 3200;
					END_IF
				
				3200:	
					IF FirstSensorOfLowerConveyor OR (NOT SecondSensorOfLowerConveyor) THEN
						LowerConveyor.M_MoveBackward();
						tonTimeOut.IN:=FALSE;
						uiBothStep := 3300;
					ELSE 
						uiBothStep := 9000;
					END_IF
					tonTimeOut.IN:=TRUE;
					IF tonTimeOut.Q=TRUE THEN
						strStatus :='Empty Robot timeout';
						_Error:=TRUE;
					END_IF	
				3300:
					IF Input.bLowCV_Block2Detect_Sensor THEN
						TON_DelayLowerCV.IN := TRUE;
					END_IF
					IF TON_DelayLowerCV.Q THEN
						LowerConveyor.M_MotorStop();
						uiBothStep := 3400;
					END_IF
				
				3400:
					TON_DelayLowerCV.IN :=FALSE;
					IF 	LowerConveyor.InStopped THEN
						tonTimeOut.IN:=FALSE;
						uiBothStep:=9000;
					END_IF
					tonTimeOut.IN:=TRUE;
					IF tonTimeOut.Q=TRUE THEN
						strStatus :='Stop Robot timeout';
						_Error:=TRUE;
					END_IF		
				9000:
						BoxReady_2nd:=TRUE;
						uiBothStep:=9999;
				
				9999: //Wait		
        // wait reset
        END_CASE

       	  // Robot Abs move
           		 Robot.M_StartRobotAbsMove( GetBox:=Get,
											UseClampA:=UseA,
											UseClampB:=UseB,
											Area:=Area,
											ClampA_Address:=Address_A,
											ClampB_Address:=Address_B,
											BoxReady_1:=BoxReady_1st,
											BoxReady_2:=BoxReady_2nd);	
		
		
        IF Robot._DI1.Done THEN
            uiExecutingStep := 30080;
        END_IF
		
    30080: // Check robot command is clear
        
        Robot.M_ResetRobotAbsMove(UseA,UseB);

        IF NOT Robot._DI1.Done THEN
			tonTimeOut.IN:=FALSE;
            uiExecutingStep := 40000; // go to place step
        END_IF    
   		//tonTimeOut.IN:=TRUE;
		IF tonTimeOut.Q=TRUE THEN
			strStatus :='Stop Robot timeout';
			_Error:=TRUE;
		END_IF

	40000:  //check the box is full ## Edit BY MIN 20250416
			 
			IF Input.bLowCV_Block2Detect_Sensor THEN 
				_Error := TRUE;
				strStatus :='LowerCV the box behind is full, please remove it';
			ELSE 
				uiExecutingStep := 40100;
			END_IF	
	
	40100:
			IF  FirstSensorOfLowerConveyor OR (NOT SecondSensorOfLowerConveyor) THEN
				tonTimeOut.IN:=FALSE;
				LowerConveyor.M_MoveBackward();
				uiExecutingStep:=40200;
			ELSE
				uiExecutingStep:=99000;
			END_IF
			tonTimeOut.IN:=TRUE;
			IF tonTimeOut.Q=TRUE THEN
				strStatus :='Lowerconveyor Reverse timeout';
				_Error:=TRUE;
			END_IF	
			
	40200:
			tonTimeOut.IN:=FALSE;
			IF Input.bLowCV_Block2Detect_Sensor THEN
				TON_DelayLowerCV.IN := TRUE;
			END_IF
			IF TON_DelayLowerCV.Q THEN
				LowerConveyor.M_MotorStop();
				uiExecutingStep := 40300;
			END_IF
			
	40300:
			IF LowerConveyor.InStopped THEN
					IF NOT (FirstSensorOfLowerConveyor) AND  SecondSensorOfLowerConveyor THEN
						uiExecutingStep := 99000;
					ELSE
						_Error := TRUE;
						strStatus := 'LowerCV the box Behind is full ,please remove it ';
					END_IF	
			END_IF
			
			tonTimeOut.IN:=TRUE;
			IF tonTimeOut.Q=TRUE THEN
				strStatus :='Lowerconveyor Reverse Stop timeout';
				_Error:=TRUE;
			END_IF
			
			
   
    99000: // process done
			TON_DelayLowerCV.IN :=FALSE;
                Status    := 'Process completed';
        		_Executed := TRUE;
END_CASE
IF _Executed THEN
    eState := STATE_DONE;
ELSIF _Error THEN
	//(iErrorID := ErrorID,UinqueErrorCode=>_UniqueErrorCode);
    eState := STATE_ERROR;
ELSIF NOT Execute THEN
    eState := STATE_RESETTING;
END_IF
IF _Abort OR Abort THEN
	//FUN_UniqueErrorCodeGenerator(iErrorID := ErrorID,UinqueErrorCode=>_UniqueErrorCode);
	eSTATE:=STATE_ABORTING;
END_IF
END_METHOD

METHOD  M_STATE_RESETTING
VAR_INPUT
END_VAR
Error :=FALSE;
Done :=FALSE;
Busy := FALSE;


CASE uiResettingStep OF
	
	0:
		tonTimeOut.IN:=FALSE;
		TON_DelayLowerCV.IN := false;
		Robot.M_ResetAllCommand();
		Robot.M_ResetRobotAbsMove(TRUE,TRUE);
		uiResettingStep:=100;
		
	100:
	
		LowerConveyor.M_MotorStop();	
		uiResettingStep:=9999;
	9999:
		_ResetCompleted:=TRUE;
END_CASE
IF _ResetCompleted THEN
	eSTATE:=STATE_DORMANT;
END_IF
END_METHOD

END_FUNCTION_BLOCK

// ---- Library/20_MachineUnits/21_StorageArea/Service/FB_WareHouseWithRobotMove.TcPOU
FUNCTION_BLOCK FB_WareHouseWithRobotMove EXTENDS FB_ObjectBase_V2 IMPLEMENTS IBasicElement
VAR_INPUT
    Robot     : REFERENCE TO FB_FanucRobot_Basic;
    WareHouse : REFERENCE TO FB_WareHouse;
   // Command   : ST_WareHouseWithRobotMove_Command;
    Info	  : st_AutoSixAxisWarehouseParameter;
	Stop	  : BOOL;
END_VAR
VAR_OUTPUT
  // Status : ST_WareHouseWithRobotMove_Status;
END_VAR
VAR
	_Abort		: BOOL;
	strStatus	: STRING;
	uiResumeStep : UINT;
	ClampA_WareHouseCoordinates : ST_WareHouseCoordinates;
    ClampB_WareHouseCoordinates : ST_WareHouseCoordinates;
	UseA 	: BOOL;
	UseB	: BOOL;
	TargetWarehouse : E_WareHouse;
	Get 	:BOOL;
	tonTimeout		:TON;
	tonRobotTimeout		:TON;
	_UniqueErrorCode :STRING;
	PreviousStrStatus : STRING;
	PreviousErrorCode : STRING;
END_VAR

SUPER^.A10_StateControl();
A00_BasicUnits();

ACTION A00_BasicUnits:
tonTimeout(PT:=T#25S);
tonRobotTimeout(PT:=T#300S);
ErrorID :=2400;
END_ACTION

METHOD M_CheckCommand : BOOL // True : Command is useful
VAR_INPUT
END_VAR
VAR
	
END_VAR
// Check command paremeter is correct

IF NOT Info.Warehouse_A AND NOT Info.Warehouse_B THEN
	strStatus:='Wrong command , No warehouse selected';
	M_CheckCommand:=FALSE;
	RETURN;
ELSIF  Info.Warehouse_A AND  Info.Warehouse_B THEN
	strStatus:='Wrong command , Both warehouses selected';
	M_CheckCommand:=FALSE;
	RETURN;
ELSIF	Info.Warehouse_A THEN
	TargetWarehouse:=E_WareHouse.WareHouseA;
ELSIF	Info.Warehouse_B THEN
	TargetWarehouse:=E_WareHouse.WareHouseB;
END_IF

IF Info.Get_A <> Info.Get_B THEN
	strStatus:='Wrong command ,GetA not match to GetB';
	M_CheckCommand:=FALSE;
	RETURN;
	ELSE
		
	Get :=Info.Get_A;
END_IF


CASE LREAL_TO_INT(Info.Layer_A) OF

1,2,3,4,5,6,7,8,9,10:
	//Normal
	// Layer A in correct range
	IF ((Info.Slide_A < 1) OR (Info.Slide_A > 20)) THEN
		strStatus := 'Command error : Clamp A target slide out of range';
		M_CheckCommand:=FALSE;
		RETURN;
	ELSE
		ClampA_WareHouseCoordinates.Layer:=LREAL_TO_INT(Info.Layer_A);
		ClampA_WareHouseCoordinates.Slide:=LREAL_TO_INT(Info.Slide_A);
   
		UseA:=TRUE;	
	END_IF
	
99:
	UseA:=FALSE;
ELSE
	 strStatus := 'Command error : Clamp A target layer out of range.';
	 M_CheckCommand:=FALSE;
	 RETURN;
END_CASE


CASE LREAL_TO_INT(Info.Layer_B) OF

1,2,3,4,5,6,7,8,9,10:
//Normal
	// Layer A in correct range
	IF ((Info.Slide_B < 1) OR (Info.Slide_B > 20)) THEN
		strStatus := 'Command error : Clamp B target slide out of range';
		M_CheckCommand:=FALSE;
		RETURN;
	ELSE
		ClampB_WareHouseCoordinates.Layer:=LREAL_TO_INT(Info.Layer_B);
		ClampB_WareHouseCoordinates.Slide:=LREAL_TO_INT(Info.Slide_B);
		UseB:=TRUE;	
	END_IF
	
99:
		UseB:=FALSE;
ELSE
	 strStatus := 'Command error : Clamp B target layer out of range.';
	 M_CheckCommand:=FALSE;
	 RETURN;
END_CASE


M_CheckCommand:=TRUE;
END_METHOD

METHOD M_CheckUnitsNotBusy : BOOL
VAR_INPUT
END_VAR
M_CheckUnitsNotBusy := true;
END_METHOD

METHOD M_CheckUnitsReady : BOOL
VAR_INPUT
END_VAR
M_CheckUnitsReady := true;
END_METHOD

METHOD  M_STATE_ABORTED
VAR_INPUT
END_VAR
ERROR :=TRUE;
Busy    := FALSE;
Aborted := TRUE;
Status := strStatus;
UniqueErrorCode:=_UniqueErrorCode;
IF NOT Execute THEN
	eSTATE:=STATE_RESETTING;
END_IF

IF Execute AND Reset THEN
	PreviousStrStatus := strStatus;
	PreviousErrorCode := _UniqueErrorCode;
	uiExecutingStep :=uiResumeStep;
	eSTATE:=STATE_EXECUTING;
END_IF
END_METHOD

METHOD  M_STATE_ABORTING
VAR_INPUT
END_VAR
CASE uiAbortingStep OF
	0 :
		uiAbortingStep:=9999;
		IF strStatus = PreviousStrStatus THEN
			_UniqueErrorCode :=PreviousErrorCode;
		END_IF
		_Abort :=FALSE;
	9999:	_AbortCompleted:=TRUE;
END_CASE

IF _AbortCompleted THEN	
	eSTATE :=STATE_ABORTED;
END_IF
END_METHOD

METHOD  M_STATE_DONE
VAR_INPUT
END_VAR
Busy := FALSE;
Done := TRUE;
IF NOT Execute THEN
    eState := STATE_RESETTING;
END_IF
END_METHOD

METHOD  M_STATE_DORMANT
VAR_INPUT
END_VAR
// Clear FB output
Busy            := FALSE;
Done            := FALSE;
Aborted         := FALSE;
Error           := FALSE;
ErrorID         := 0;
Status          := '';
_ResetCompleted := FALSE;
_Error          := FALSE;
_Executed       := FALSE;
strStatus :='No Error';
tonTimeout.IN :=FALSE;
tonRobotTimeout.IN :=FALSE;
uiExecutingStep :=uiResettingStep :=uiResumeStep :=0;
PreviousStrStatus			 :='';
PreviousErrorCode			 :='';

// Wait Execute command
IF Execute THEN
    eState := STATE_EXECUTING;
END_IF
END_METHOD

METHOD  M_STATE_ERROR
VAR_INPUT
END_VAR
ERROR   :=TRUE;
Busy	:=FALSE;
Status := strStatus;
UniqueErrorCode:=_UniqueErrorCode;
IF NOT Execute THEN	
eSTATE:=STATE_RESETTING;
END_IF
END_METHOD

METHOD  M_STATE_EXECUTING
VAR_INPUT
END_VAR
VAR_INST
	BoxReady_1st : BOOL;
	BoxReady_2nd : BOOL;  
    uiBothStep : UINT;
    ClampA_WareHouseCoordinates : ST_WareHouseCoordinates;
    ClampB_WareHouseCoordinates : ST_WareHouseCoordinates;
	

	
END_VAR
VAR
	
END_VAR
// Set Busy active edit by johnson
Busy := TRUE;
IF THIS^.Stop THEN // Pending the timeout when Stop signal occur
	tonTimeout.IN :=FALSE;
	tonRobotTimeout.IN :=FALSE;
END_IF
// Service Process
CASE uiExecutingStep OF
	0:
        // Clear variable
       
        tonTimeout.IN :=FALSE;
        uiBothStep := 0;
		BoxReady_1st := 0;
		BoxReady_2nd := 0;
        // Check command
        IF M_CheckCommand() THEN
            uiExecutingStep := 10;
		ELSE
			_Error:=TRUE;
        END_IF
    10:
        // Start process, check units first
        IF M_CheckUnitsReady() THEN
            uiExecutingStep := 20;
        END_IF
    20:
        // CHeck units not busy state
        IF M_CheckUnitsNotBusy() THEN
            uiExecutingStep := 1000;
        END_IF
   
	1000:   
			// Read  Warehouse coordinate
			ClampA_WareHouseCoordinates := THIS^.ClampA_WareHouseCoordinates;
            ClampB_WareHouseCoordinates := THIS^.ClampB_WareHouseCoordinates;     
			IF UseA AND NOT UseB THEN
				//Only clampA
				uiExecutingStep := 10000;
			ELSIF NOT UseA AND UseB THEN
				//Only ClampB 
				uiExecutingStep := 20000;
			ELSIF UseA AND UseB THEN
				//Both Clamps
				uiExecutingStep := 30000;		
			END_IF
       
    10000: // Only ClampA 
        IF NOT Robot._DI1.Done THEN
            // Read ClampA Warehouse coordinate
            ClampA_WareHouseCoordinates := THIS^.ClampA_WareHouseCoordinates;
			
			IF Get THEN// Prepare Box
				//Pick Box
				 WareHouse.M_StartReloadBox(WareHouseSelect := TargetWarehouse, WarehouseCoordinates := ClampA_WareHouseCoordinates);

           		 // Check Box reload completed
           		 IF WareHouse.bReloadBox_Completed THEN
           	     BoxReady_1st := TRUE;
          		  END_IF
				  // Robot Warehouse move
           		 Robot.M_StartWareHousePickUpBox_ClampA(WareHouseSelect := TargetWarehouse,
                                                   Info            := ClampA_WareHouseCoordinates,
                                                   BoxReady_1st    := BoxReady_1st);
				tonTimeout.IN:=TRUE;
				IF tonTimeout.Q THEN
					_Error:=TRUE;
					strStatus:='Clamp A reolad box timeout';
				END_IF
				  
			ELSE
					//Place Box
					WareHouse.M_StartFeedInBox(WareHouseSelect := TargetWarehouse, WarehouseCoordinates := ClampA_WareHouseCoordinates);

           			 // Check Box reload completed
           			 IF WareHouse.bFeedInBox_Completed THEN
               			 BoxReady_1st := TRUE;
          		 	 END_IF				
					           
			 	Robot.M_StartWareHousePlaceBox_ClampA(WareHouseSelect := TargetWarehouse,
                                                   Info            := ClampA_WareHouseCoordinates,
                                                   BoxReady_1st    := BoxReady_1st);
            	
				tonTimeout.IN:=TRUE;
				IF tonTimeout.Q THEN
					_Error:=TRUE;
					strStatus:='Clamp A Feedin box timeout';
				END_IF
           END_IF
        ELSE
            uiExecutingStep := 10080;
        END_IF
		
		tonRobotTimeout.IN :=TRUE;
		IF tonRobotTimeout.Q THEN
			_Error:=TRUE;
			strStatus:='Clamp A  robot timeout';
		END_IF
		
    10080:
        Robot.M_ResetAllCommand(); // Clear command and go to place box
		tonTimeout.IN :=FALSE;
		tonRobotTimeout.IN :=FALSE;
        IF NOT Robot._DI1.Done THEN
            uiExecutingStep := 99000; 
        END_IF
    
    
   20000: // Only ClampB
        IF NOT Robot._DI1.Done THEN
            			
			IF Get THEN// Prepare Box
				//Pick Box
				 WareHouse.M_StartReloadBox(WareHouseSelect := TargetWarehouse, WarehouseCoordinates := ClampB_WareHouseCoordinates);

           		 // Check Box reload completed
           		 IF WareHouse.bReloadBox_Completed THEN
           	     BoxReady_2nd := TRUE;
          		  END_IF
				  // Robot Warehouse move
           		 Robot.M_StartWareHousePickUpBox_ClampB(WareHouseSelect := TargetWarehouse,
                                                   Info            := ClampB_WareHouseCoordinates,
                                                   BoxReady_2nd    := BoxReady_2nd);

				tonTimeout.IN:=TRUE;
				IF tonTimeout.Q THEN
					_Error:=TRUE;
					strStatus:='Clamp B Reload box timeout';
				END_IF
			ELSE
					//Place Box
					WareHouse.M_StartFeedInBox(WareHouseSelect := TargetWarehouse, WarehouseCoordinates := ClampB_WareHouseCoordinates);

           			 // Check Box reload completed
           			 IF WareHouse.bFeedInBox_Completed THEN
               			 BoxReady_2nd := TRUE;
          		 	 END_IF				
					           
			 	Robot.M_StartWareHousePlaceBox_ClampB (WareHouseSelect := TargetWarehouse,
                                                   Info            := ClampB_WareHouseCoordinates,
                                                   BoxReady_2nd    := BoxReady_2nd);
            	tonTimeout.IN:=TRUE;
				IF tonTimeout.Q THEN
					_Error:=TRUE;
					strStatus:='Clamp B Feedin box timeout';
				END_IF
           END_IF
        ELSE
            uiExecutingStep := 20080;
        END_IF
		tonRobotTimeout.IN :=TRUE;
		IF tonRobotTimeout.Q THEN
			_Error:=TRUE;
			strStatus:='Clamp B Robot timeout';
		END_IF
		
    20080:
        Robot.M_ResetAllCommand(); // Clear command and go to place box
		tonTimeout.IN :=FALSE;
		tonRobotTimeout.IN :=FALSE;

        IF NOT Robot._DI1.Done THEN
            uiExecutingStep := 99000; 
        END_IF
		
    30000: // Both Clamps
        		
		IF Get THEN //BOth clamps pick
        CASE uiBothStep OF
            0: // ClampA target slide move the box to front side
                WareHouse.M_StartReloadBox(WareHouseSelect      := TargetWarehouse,
                                           WarehouseCoordinates := ClampA_WareHouseCoordinates);
				
				tonTimeout.IN :=TRUE;
				IF tonTimeout.Q THEN
					_Error:=TRUE;
					strStatus:='Clamp A reload timeout';
				END_IF
               
                IF WareHouse.bReloadBox_Completed THEN
					tonTimeout.IN :=FALSE;
                    BoxReady_1st     := TRUE;
                    uiBothStep := 10;
                END_IF

            10: // wait Robot Allow continue
			 		WareHouse.M_ResetReloadBox();
                IF Robot._DI1.Notification // AND
//                    NOT
//                    WareHouse._stWarehouseList.ASide_Layers[ClampA_WareHouseCoordinates.Layer].stStatus.bSlides[ClampA_WareHouseCoordinates.Slide]
                    THEN
                   
					
                    IF NOT WareHouse.bReloadBox_Completed THEN					
               
                        uiBothStep := 15;
                    END_IF

                END_IF
			15:	IF NOT WareHouse._stWarehouseList.ASide_Layers[ClampA_WareHouseCoordinates.Layer].stStatus.bSlides[ClampA_WareHouseCoordinates.Slide] THEN
					 uiBothStep := 20;	
				 END_IF
				 
            20: // ClampB target slide move the box to front slide
                WareHouse.M_StartReloadBox(WareHouseSelect := TargetWarehouse, WarehouseCoordinates := ClampB_WareHouseCoordinates);
				tonTimeout.IN :=TRUE;
                IF WareHouse.bReloadBox_Completed THEN
					tonTimeout.IN :=FALSE;
                    BoxReady_2nd     := TRUE;
                    uiBothStep := 99;
                END_IF
				IF tonTimeout.Q THEN
					_Error:=TRUE;
					strStatus:='Clamp B reload timeout';
				END_IF
				
				
            99:
				WareHouse.M_ResetReloadBox();
        // wait reset
        END_CASE

        Robot.M_StartWareHousePickUpBox_ClampBoth(WareHouseSelect := TargetWarehouse,
                                                  ClampA_Info     := ClampA_WareHouseCoordinates,
                                                  ClampB_Info     := ClampB_WareHouseCoordinates,
                                                  BoxReady_1st    := BoxReady_1st,
                                                  BoxReady_2nd    := BoxReady_2nd);
												  
		tonRobotTimeout.IN :=TRUE;
		IF tonRobotTimeout.Q THEN
			_Error:=TRUE;
			strStatus:='Robot timeout';
		END_IF
		ELSE
		  CASE uiBothStep OF
			  
			   0: // ClampA target slide move the box to front side
                WareHouse.M_StartFeedInBox(WareHouseSelect      := TargetWarehouse,
                                           WarehouseCoordinates := ClampA_WareHouseCoordinates);

               tonTimeout.IN :=TRUE;
                IF WareHouse.bFeedInBox_Completed THEN
					tonTimeout.IN :=FALSE;
                    BoxReady_1st     := TRUE;
                    uiBothStep := 10;
                END_IF
				IF tonTimeout.Q THEN
					_Error:=TRUE;
					strStatus:='Clamp A Feedin timeout';
				END_IF

            10: // wait Robot Allow continue
					WareHouse.M_ResetFeedInBox();
                 IF Robot._DI1.Notification //AND
                     
//                    WareHouse._stWarehouseList.ASide_Layers[ClampA_WareHouseCoordinates.Layer].stStatus.bSlides[ClampA_WareHouseCoordinates.Slide]
                    THEN
                    

                    IF NOT WareHouse.bFeedInBox_Completed THEN
                        uiBothStep := 15;
                    END_IF

                END_IF
			15:  
				uiBothStep := 20;
			
            20: // ClampB target slide move the box to front slide
                WareHouse.M_StartFeedInBox(WareHouseSelect := TargetWarehouse, WarehouseCoordinates := ClampB_WareHouseCoordinates);
				tonTimeout.IN :=TRUE;
                IF WareHouse.bFeedInBox_Completed THEN
					tonTimeout.IN :=FALSE;
                    BoxReady_2nd     := TRUE;
                    uiBothStep := 99;
                END_IF
				IF tonTimeout.Q THEN
					_Error:=TRUE;
					strStatus:='Clamp B Feedin timeout';
				END_IF
            99: 
				WareHouse.M_ResetFeedInBox();

        END_CASE

        Robot.M_StartWareHousePlaceUpBox_ClampBoth(WareHouseSelect := TargetWarehouse,
                                                  ClampA_Info     := ClampA_WareHouseCoordinates,
                                                  ClampB_Info     := ClampB_WareHouseCoordinates,
                                                  BoxReady_1st    := BoxReady_1st,
                                                  BoxReady_2nd    := BoxReady_2nd);
												  
		tonRobotTimeout.IN :=TRUE;
		IF tonRobotTimeout.Q THEN
			_Error:=TRUE;
			strStatus:='Robot timeout';
		END_IF
		END_IF
		
        IF Robot._DI1.Done THEN
            uiExecutingStep := 30080;
        END_IF
		
    30080: // Check robot command is clear
        WareHouse.M_ResetReloadBox();
        WareHouse.M_ResetFeedInBox();
        Robot.M_ResetAllCommand();
		tonTimeout.IN :=FALSE;
		tonRobotTimeout.IN :=FALSE;
		
        IF NOT Robot._DI1.Done THEN
            uiExecutingStep := 99000; // go to place step
        END_IF    
   
   
    99000: // process done
                Status    := 'Process completed';
        _Executed := TRUE;
END_CASE
IF _Executed THEN
    eState := STATE_DONE;
ELSIF _Error THEN
	//FUN_UniqueErrorCodeGenerator(iErrorID := ErrorID,UinqueErrorCode=>_UniqueErrorCode);
    eState := STATE_ERROR;
ELSIF NOT Execute THEN
    eState := STATE_RESETTING;
END_IF
IF _Abort OR Abort THEN
	//FUN_UniqueErrorCodeGenerator(iErrorID := ErrorID,UinqueErrorCode=>_UniqueErrorCode);
	eSTATE:=STATE_ABORTING;
END_IF
END_METHOD

METHOD  M_STATE_RESETTING
VAR_INPUT
END_VAR
Error :=FALSE;
Done :=FALSE;
Busy := FALSE;
_Error :=FALSE;

CASE uiResettingStep OF
	
	0:
		tonTimeout.IN :=FALSE;
		Robot.M_ResetAllCommand();
		uiResettingStep:=9999;
		WareHouse.M_ResetFeedInBox();
		WareHouse.M_ResetReloadBox();
	9999:
		_ResetCompleted:=TRUE;
END_CASE
IF _ResetCompleted THEN
	eSTATE:=STATE_DORMANT;
END_IF
END_METHOD

END_FUNCTION_BLOCK

// ---- Library/20_MachineUnits/21_StorageArea/Service/FB_StorageHoming.TcPOU
FUNCTION_BLOCK FB_StorageHoming EXTENDS FB_ActionBasic
VAR_INPUT
	xExecute : BOOL;
	xAbort : BOOL;
    Cylinder   : REFERENCE TO UNI_CylinderList;
    Motor      : REFERENCE TO UNI_MotorList;
    FanucRobot : REFERENCE TO FB_FanucRobot_Basic;
	Homed : REFERENCE TO BOOL;
END_VAR
VAR_OUTPUT
	xAborted : BOOL;
	iErrorID : INT;
	ErrorMsg : STRING;
	RobotResetCMD : BOOL;
	RackMotorHomeRequest : BOOL;
END_VAR
VAR
	StateBehaviour : CBML.ETrigA;
	uiStorageHomingStep : UINT;
	CylinderCheckTon : TON;
	MotorCheckTon : TON;
	FanucRobotCheckTon : TON;
	ResetRobotDelay	 	: TON ;
	fbExecuteEdgeDetect :FB_EdgeDetect;
END_VAR

THIS^.IBehaviourModel := StateBehaviour;
StateBehaviour(xExecute := xExecute,
    xDone => xDone,
    xBusy => xBusy,
    xError => xError,
    xAbort := xAbort OR fbExecuteEdgeDetect.xFallingEdge,
    xAborted => xAborted);

//Error Msg
iErrorID := StateBehaviour._model.iErrorID;
ErrorMsg := M_GetErrorMsg(xErrorID := iErrorID);

//Make sure that C# turns off execute to shut down the service
fbExecuteEdgeDetect(xInput :=xExecute);


CylinderCheckTon(PT := T#5S);
MotorCheckTon(PT := T#2S);
FanucRobotCheckTon(PT:=T#60S);
ResetRobotDelay(PT:=T#300ms);

METHOD CleanupAction
VAR_INPUT
    xAbortProposed : BOOL;
    iErrorIDProposed: INT;
END_VAR
VAR_OUTPUT
    xComplete : BOOL := TRUE;
    xAbort: BOOL := xAbortProposed;
 	iErrorID : INT := iErrorIDProposed;
END_VAR
END_METHOD

METHOD CyclicAction
VAR_INPUT
    itfTimingController : CBML.ITimingController;
END_VAR
VAR_OUTPUT
    xComplete : BOOL := TRUE;
    iErrorID : INT := 0;
END_VAR
VAR
	tehn: INT;
END_VAR
xComplete := FALSE;
CASE uiStorageHomingStep OF
	0: // Retract Cylinder
		M_RetractStorageCylinder();
		RobotResetCMD := FALSE;	
		Cylinder.List.fbStackPush.M_Retract();
		IF Cylinder.List.fbStackPush.InRearPosition THEN		// safecheck Rackmotor home 
		uiStorageHomingStep := 100;
		END_IF
	100:
		IF M_CheckStorageCylinderInRear() THEN
			uiStorageHomingStep := 200;
		ELSE
			CylinderCheckTon.IN := TRUE;
			IF CylinderCheckTon.Q THEN
				iErrorID := 2;
			END_IF
		END_IF
	200:
			CylinderCheckTon.IN := FALSE;
			M_StopStorageMotor ();
			uiStorageHomingStep := 300;
	300:
		IF M_CheckStorageMotorInStop() THEN
			uiStorageHomingStep := 400;
		ELSE
			MotorCheckTon.IN := TRUE;
			IF MotorCheckTon.Q THEN
				iErrorID := 3;
			END_IF
		END_IF
	400:
		MotorCheckTon.IN := FALSE;
		FanucRobotCheckTon.IN := TRUE;
		IF FanucRobot.Error THEN
			RobotResetCMD := TRUE;		
			ResetRobotDelay.IN:=TRUE;
		ELSE
			uiStorageHomingStep := 500;
		END_IF
		IF ResetRobotDelay.Q THEN
			ResetRobotDelay.IN:=FALSE;
			uiStorageHomingStep := 500;
		END_IF	
		
		
	500:
		RobotResetCMD := FALSE;	
		RackMotorHomeRequest := TRUE;		// RackMotor homing edit min
		FanucRobot.OpMode := E_FanucRobotOpMode.RSR02;
		IF FanucRobot.Error THEN
			RobotResetCMD := TRUE;		
		END_IF
		IF FanucRobot._RSR2_Completed THEN
			uiStorageHomingStep := 600;
		END_IF
	600:
		FanucRobot.OpMode := E_FanucRobotOpMode.RSR01;
		IF FanucRobot._RSR1_Ready THEN
			uiStorageHomingStep := 700;
		END_IF
	700:
		FanucRobotCheckTon.IN := FALSE;
		Homed := TRUE;
		xComplete := TRUE;
END_CASE

IF FanucRobotCheckTon.Q THEN
	iErrorID := 4;
END_IF
END_METHOD

METHOD ExitAction
VAR_INPUT
    xAfterCleanup : BOOL;
    xInCopyCode : BOOL;
END_VAR
uiStorageHomingStep := 0;
END_METHOD

METHOD M_CheckStorageCylinderInRear : BOOL
VAR_INPUT
END_VAR
M_CheckStorageCylinderInRear := Cylinder.List.fbUpCV_FeedInPress1.InRearPosition AND
    Cylinder.List.fbUpCV_FeedInPress2.InRearPosition AND
    Cylinder.List.fbUpCV_DiameterPress.InRearPosition AND
    Cylinder.List.fbUpCV_CamaraPress1.InRearPosition AND
    Cylinder.List.fbUpCV_CamaraPress2.InRearPosition AND
    Cylinder.List.fbUpCV_CamaraPress3.InRearPosition AND
    Cylinder.List.fbUpCV_CamaraPress4.InRearPosition AND
    Cylinder.List.fbUpCV_Block1.InRearPosition AND
    Cylinder.List.fbUpCV_Block2.InRearPosition AND
    Cylinder.List.fbUpCV_Block3.InRearPosition AND
    Cylinder.List.fbUpCV_DiameterHoriz.InRearPosition AND
    Cylinder.List.fbUpCV_DiameterVert.InRearPosition AND
    Cylinder.List.fbUpCV_DiameterClamp.InRearPosition AND
    Cylinder.List.fbStackPush.InRearPosition AND
    Cylinder.List.fbLowCV_Press1.InRearPosition AND
    Cylinder.List.fbLowCV_Press2.InRearPosition AND
    Cylinder.List.fbLowCV_Press3.InRearPosition AND
    Cylinder.List.fbLowCV_Press4.InRearPosition AND
    Cylinder.List.fbLowCV_Block1.InRearPosition AND
    Cylinder.List.fbLowCV_Block2.InRearPosition;
END_METHOD

METHOD M_CheckStorageMotorInStop : BOOL
VAR_INPUT
END_VAR
M_CheckStorageMotorInStop := Motor.List.LowCV.InStopped AND
    Motor.List.UpCV.InStopped AND
    Motor.List.WareHouseCV_01.InStopped AND
    Motor.List.WareHouseCV_02.InStopped AND
    Motor.List.WareHouseCV_03.InStopped AND
    Motor.List.WareHouseCV_04.InStopped AND
    Motor.List.WareHouseCV_05.InStopped AND
    Motor.List.WareHouseCV_06.InStopped AND
    Motor.List.WareHouseCV_07.InStopped AND
    Motor.List.WareHouseCV_08.InStopped AND
    Motor.List.WareHouseCV_09.InStopped AND
    Motor.List.WareHouseCV_10.InStopped AND
    Motor.List.WareHouseCV_11.InStopped AND
    Motor.List.WareHouseCV_12.InStopped AND
    Motor.List.WareHouseCV_13.InStopped AND
    Motor.List.WareHouseCV_14.InStopped AND
    Motor.List.WareHouseCV_15.InStopped AND
    Motor.List.WareHouseCV_16.InStopped AND
    Motor.List.WareHouseCV_17.InStopped AND
    Motor.List.WareHouseCV_18.InStopped AND
    Motor.List.WareHouseCV_19.InStopped AND
    Motor.List.WareHouseCV_20.InStopped;
END_METHOD

METHOD M_GetErrorMsg : T_MaxString
VAR_INPUT
	xErrorID: INT;
END_VAR

VAR
	
END_VAR
CASE xErrorID OF
    0:
        M_GetErrorMsg := 'No Error';
    1:
        M_GetErrorMsg := 'Action time out';
    2:
        M_GetErrorMsg := 'Cylinder not ready';
    3:
        M_GetErrorMsg := 'Motor not ready';
    4:
		M_GetErrorMsg := 'FanucRobot can not homing';
END_CASE
END_METHOD

METHOD M_RetractStorageCylinder : BOOL
VAR_INPUT
END_VAR
Cylinder.List.fbUpCV_FeedInPress1.M_Retract();
Cylinder.List.fbUpCV_FeedInPress2.M_Retract();
Cylinder.List.fbUpCV_DiameterPress.M_Retract();
Cylinder.List.fbUpCV_CamaraPress1.M_Retract();
Cylinder.List.fbUpCV_CamaraPress2.M_Retract();
Cylinder.List.fbUpCV_CamaraPress3.M_Retract();
Cylinder.List.fbUpCV_CamaraPress4.M_Retract();
Cylinder.List.fbUpCV_Block1.M_Retract();
Cylinder.List.fbUpCV_Block2.M_Retract();
Cylinder.List.fbUpCV_Block3.M_Retract();
Cylinder.List.fbUpCV_DiameterHoriz.M_Retract();
Cylinder.List.fbUpCV_DiameterVert.M_Retract();
Cylinder.List.fbUpCV_DiameterClamp.M_Retract();
Cylinder.List.fbStackPush.M_Retract();
Cylinder.List.fbLowCV_Press1.M_Retract();
Cylinder.List.fbLowCV_Press2.M_Retract();
Cylinder.List.fbLowCV_Press3.M_Retract();
Cylinder.List.fbLowCV_Press4.M_Retract();
Cylinder.List.fbLowCV_Block1.M_Retract();
Cylinder.List.fbLowCV_Block2.M_Retract();

M_RetractStorageCylinder := TRUE;
END_METHOD

METHOD M_StopStorageMotor : BOOL
VAR_INPUT
END_VAR
Motor.List.LowCV.M_MotorStop();
Motor.List.UpCV.M_MotorStop();
Motor.List.WareHouseCV_01.M_MotorStop();
Motor.List.WareHouseCV_02.M_MotorStop();
Motor.List.WareHouseCV_03.M_MotorStop();
Motor.List.WareHouseCV_04.M_MotorStop();
Motor.List.WareHouseCV_05.M_MotorStop();
Motor.List.WareHouseCV_06.M_MotorStop();
Motor.List.WareHouseCV_07.M_MotorStop();
Motor.List.WareHouseCV_08.M_MotorStop();
Motor.List.WareHouseCV_09.M_MotorStop();
Motor.List.WareHouseCV_10.M_MotorStop();
Motor.List.WareHouseCV_11.M_MotorStop();
Motor.List.WareHouseCV_12.M_MotorStop();
Motor.List.WareHouseCV_13.M_MotorStop();
Motor.List.WareHouseCV_14.M_MotorStop();
Motor.List.WareHouseCV_15.M_MotorStop();
Motor.List.WareHouseCV_16.M_MotorStop();
Motor.List.WareHouseCV_17.M_MotorStop();
Motor.List.WareHouseCV_18.M_MotorStop();
Motor.List.WareHouseCV_19.M_MotorStop();
Motor.List.WareHouseCV_20.M_MotorStop();

M_StopStorageMotor := TRUE;
END_METHOD

METHOD ResetAction
VAR_OUTPUT
    xComplete : BOOL := TRUE;
END_VAR
uiStorageHomingStep := 0;
RobotResetCMD := FALSE;
CylinderCheckTon.IN := FALSE;
MotorCheckTon.IN := FALSE;
FanucRobotCheckTon.IN := FALSE;
RackMotorHomeRequest := false;
END_METHOD

METHOD StartAction
VAR_OUTPUT
    xComplete : BOOL := TRUE;
	iErrorID : INT := 0;
END_VAR

VAR
	uiCylinderIndex :UINT;
	uiMotorIndex : UINT;
END_VAR
Homed := FALSE;
RackMotorHomeRequest := false;
ResetRobotDelay.IN := FALSE;
uiStorageHomingStep := 0;
END_METHOD

END_FUNCTION_BLOCK

// ---- Library/20_MachineUnits/21_StorageArea/Service/FB_DiameterMovement.TcPOU
FUNCTION_BLOCK FB_DiameterMovement EXTENDS FB_ObjectBase_V2
VAR_INPUT
//    Execute    :BOOL;   // True : This prog will start.
//    Abort      :BOOL;   // True : This prog will be abort.
//    Reset      :BOOL;   // True : This prog will be reset.
//    ObjectName :STRING; // Set this fb name(About it's action)
	
	bContinue:BOOL;
	
//	DiameterHorizontalCylinder 	:REFERENCE TO FB_Cylinder;	//測徑橫移氣壓缸
//	DiameterUpDownCylinder		:REFERENCE TO FB_Cylinder;	//測徑上下氣壓缸
//	DiameterClampCylinder		:REFERENCE TO FB_Cylinder; //測徑夾爪氣壓缸

	Cylinder : REFERENCE TO UNI_CylinderList;
	
END_VAR

VAR_OUTPUT
//    Busy    :BOOL;        // True : This prog is running.
//    Done    :BOOL;        // True : Command has been executed.
//    Aborted :BOOL;        // True : This prog is aborted.
//    Error   :BOOL;        // True : This prog has an error.
//    ErrorID :UINT;       // Output ErrorID
//    Status  :T_MaxString; // Output this prog status by string(255bytes)
	PickDone	:BOOL;
END_VAR

VAR
//    eState :E_MethodStatus_Basic;
//	uiExecutingStep : UDINT; // This var is used to been controll STATE_EXECUTING process.
//	uiResettingStep : UDINT;
//	uiAbortingStep : UDINT;
//	_Executed :BOOL; // Executing process completed.
//	_Error : BOOL; // FB has an error.
//	_ResetCompleted : BOOL; // FB resetting completed.
//	_AbortCompleted : BOOL; // FB aborting completed.
	_Abort		: BOOL;
	strStatus	: STRING;
	uiResumeStep : UINT;
	tonDiameterTimeoutTwo :TON;
	
END_VAR

A00_BasicUnits();
SUPER^.A10_StateControl();

ACTION A00_BasicUnits:
tonDiameterTimeoutTwo(PT:=T#2S);
END_ACTION

METHOD GetModelState
VAR_OUTPUT
    xDone    :BOOL;
    xBusy    :BOOL;
    xError   :BOOL;
    xAborted :BOOL;
    iErrorID :UDINT;
	UniqueErrorCode : STRING;
END_VAR
xDone    := Done;
xBusy    := Busy;
xError   := Error;
xAborted := Abort;
iErrorID := ErrorID;
END_METHOD

METHOD GetName : STRING
GetName := ObjectName;
END_METHOD

METHOD  M_STATE_ABORTED
VAR_INPUT
END_VAR
ERROR :=TRUE;
Status := strStatus;

IF NOT Execute THEN
	eSTATE:=STATE_RESETTING;
END_IF

IF Execute AND Reset THEN
	uiExecutingStep :=uiResumeStep;
	eSTATE:=STATE_EXECUTING;
END_IF
END_METHOD

METHOD  M_STATE_ABORTING
VAR_INPUT
END_VAR
CASE uiAbortingStep OF
	
	
	9999:	_AbortCompleted:=TRUE;
END_CASE

IF _AbortCompleted THEN	
	eSTATE :=STATE_ABORTED;
END_IF
END_METHOD

METHOD  M_STATE_DONE
VAR_INPUT
END_VAR
Busy := FALSE;
Done:=TRUE;

IF NOT Execute THEN
	eSTATE:=STATE_RESETTING;
END_IF
END_METHOD

METHOD  M_STATE_DORMANT
VAR_INPUT
END_VAR
_Executed:=FALSE;
_Error	:=FALSE;
_Abort :=FALSE;
strStatus :='No Error';
uiResettingStep:=0;
uiExecutingStep :=0;
tonDiameterTimeoutTwo.IN:=FALSE;
Error := Busy := Done := FALSE;

IF Execute THEN
	eSTATE:=STATE_EXECUTING;
END_IF
END_METHOD

METHOD  M_STATE_ERROR
VAR_INPUT
END_VAR
ERROR :=TRUE;
Busy :=FALSE;
Done := FALSE;
Status := strStatus;
IF NOT Execute THEN	
eSTATE:=STATE_RESETTING;
END_IF
END_METHOD

METHOD  M_STATE_EXECUTING
VAR_INPUT
END_VAR
Busy :=TRUE;

CASE uiExecutingStep OF
	

0: //Standby todo : check 
	
		uiExecutingStep:=10;
10:
		
		IF Cylinder.List.fbUpCV_DiameterHoriz.xError THEN
			Cylinder.List.fbUpCV_DiameterHoriz.M_Reset();
		END_IF
		IF Cylinder.List.fbUpCV_DiameterVert.xError THEN
			Cylinder.List.fbUpCV_DiameterVert.M_Reset();
		END_IF
		IF Cylinder.List.fbUpCV_DiameterClamp.xError THEN
			Cylinder.List.fbUpCV_DiameterClamp.M_Reset();
		END_IF
		uiExecutingStep:=20;
		
20:
	Cylinder.List.fbUpCV_DiameterVert.M_Retract();
	IF Cylinder.List.fbUpCV_DiameterClamp.InFrontPosition THEN
		uiExecutingStep:=30;
	ELSE
		uiExecutingStep:=60;	
	END_IF
30:
	
	IF Cylinder.List.fbUpCV_DiameterVert.InRearPosition THEN
		Cylinder.List.fbUpCV_DiameterHoriz.M_Extend();
		uiExecutingStep:=40;
	END_IF
40:		
	IF Cylinder.List.fbUpCV_DiameterHoriz.InFrontPosition THEN
		Cylinder.List.fbUpCV_DiameterClamp.M_Retract();
		uiExecutingStep:=50;
	END_IF
50:	
	IF Cylinder.List.fbUpCV_DiameterClamp.InRearPosition THEN
		uiExecutingStep:=60;
	END_IF
	
60 : 
	Cylinder.List.fbUpCV_DiameterHoriz.M_Retract();
		uiExecutingStep:=70;
70:
	IF Cylinder.List.fbUpCV_DiameterHoriz.InRearPosition THEN
		uiExecutingStep:=1000;	
	END_IF
			
	

1000:// Pick to diameter camera position start: Clamp down
	Cylinder.List.fbUpCV_DiameterVert.M_Extend();
	uiExecutingStep:=1100;
	
1100:// wait clamp down
	tonDiameterTimeoutTwo.IN:=TRUE;
	IF 	Cylinder.List.fbUpCV_DiameterVert.InFrontPosition THEN
		tonDiameterTimeoutTwo.IN:=FALSE;
		uiExecutingStep:=1200;
	END_IF
	IF tonDiameterTimeoutTwo.Q THEN
		_Error :=TRUE;
		strStatus:='Cylinder.List.fbUpCV_DiameterVert MoveForward Timeout';
	END_IF
	
1200: // Clamp close
	Cylinder.List.fbUpCV_DiameterClamp.M_Extend();
	uiExecutingStep:=1300;

1300://wait clamp close
	tonDiameterTimeoutTwo.IN:=TRUE;
	IF 	Cylinder.List.fbUpCV_DiameterClamp.InFrontPosition THEN
		tonDiameterTimeoutTwo.IN :=FALSE;
		uiExecutingStep:=1400;
	END_IF
	IF tonDiameterTimeoutTwo.Q THEN
		_Error :=TRUE;
		strStatus:='Cylinder.List.fbUpCV_DiameterClamp M_Extend Timeout';
	END_IF
1400 : //Clamp up
	Cylinder.List.fbUpCV_DiameterVert.M_Retract();
	uiExecutingStep:=1500;	

1500:// wait clamp up
		tonDiameterTimeoutTwo.IN :=TRUE;
	IF 	Cylinder.List.fbUpCV_DiameterVert.InRearPosition THEN
		tonDiameterTimeoutTwo.IN :=FALSE;
		uiExecutingStep:=1600;
	END_IF
	IF tonDiameterTimeoutTwo.Q THEN
		_Error :=TRUE;
		strStatus:='Cylinder.List.fbUpCV_DiameterVert M_Retract Timeout';
	END_IF
1600: //Move horizontal
	Cylinder.List.fbUpCV_DiameterHoriz.M_Extend();
	uiExecutingStep:=1700;

1700://wait move horizontal
		tonDiameterTimeoutTwo.IN:=TRUE;
	IF 	Cylinder.List.fbUpCV_DiameterHoriz.InFrontPosition THEN
		tonDiameterTimeoutTwo.IN :=FALSE;
		uiExecutingStep:=1800;
	END_IF
		IF tonDiameterTimeoutTwo.Q THEN
		_Error :=TRUE;
		strStatus:='Cylinder.List.fbUpCV_DiameterHoriz M_Extend Timeout';
	END_IF

1800://Move down to diameter camera position
	Cylinder.List.fbUpCV_DiameterVert.M_Extend();
	uiExecutingStep:=1900;
	
1900:
		tonDiameterTimeoutTwo.IN:=TRUE;
	IF 	Cylinder.List.fbUpCV_DiameterVert.InFrontPosition THEN
		tonDiameterTimeoutTwo.IN :=FALSE;
		uiExecutingStep:=2000;
	END_IF	
	IF tonDiameterTimeoutTwo.Q THEN
		_Error :=TRUE;
		strStatus:='Cylinder.List.fbUpCV_DiameterVert M_Extend Timeout';
	END_IF

2000: 
	PickDone :=TRUE;
	IF bContinue THEN
		PickDone :=FALSE;
		uiExecutingStep:=5000;
	END_IF

5000: // Place needle back to box start
	Cylinder.List.fbUpCV_DiameterVert.M_Retract();
	uiExecutingStep:=5100;
	
5100:// wait clamp down
	tonDiameterTimeoutTwo.IN :=TRUE;
	IF 	Cylinder.List.fbUpCV_DiameterVert.InRearPosition THEN
		tonDiameterTimeoutTwo.IN :=FALSE;
		uiExecutingStep:=5200;
	END_IF
	IF tonDiameterTimeoutTwo.Q THEN
		_Error :=TRUE;
		strStatus:='Cylinder.List.fbUpCV_DiameterVert M_Retract Timeout';
	END_IF
	
5200: 
		Cylinder.List.fbUpCV_DiameterHoriz.M_Retract();
		uiExecutingStep := 5300;

5300:
		tonDiameterTimeoutTwo.IN :=TRUE;
		IF Cylinder.List.fbUpCV_DiameterHoriz.InRearPosition THEN
			tonDiameterTimeoutTwo.IN :=FALSE;
			uiExecutingStep := 5400;
		END_IF
		IF tonDiameterTimeoutTwo.Q THEN
		_Error :=TRUE;
		strStatus:='Cylinder.List.fbUpCV_DiameterHoriz M_Retract Timeout';
		END_IF
5400 : 
		Cylinder.List.fbUpCV_DiameterVert.M_Extend();
		uiExecutingStep:=5500;

5500:
		tonDiameterTimeoutTwo.IN :=TRUE;
		IF 	Cylinder.List.fbUpCV_DiameterVert.InFrontPosition THEN
			tonDiameterTimeoutTwo.IN:=FALSE;
			uiExecutingStep:=5600;
		END_IF
		IF tonDiameterTimeoutTwo.Q THEN
		_Error :=TRUE;
		strStatus:='Cylinder.List.fbUpCV_DiameterVert M_Extend Timeout';
		END_IF
5600: 
		Cylinder.List.fbUpCV_DiameterClamp.M_Retract();
		uiExecutingStep := 5700;
5700:	
		tonDiameterTimeoutTwo.IN :=TRUE;
		IF Cylinder.List.fbUpCV_DiameterClamp.InRearPosition THEN
			tonDiameterTimeoutTwo.IN :=FALSE;
			uiExecutingStep :=5800;
		END_IF
		IF tonDiameterTimeoutTwo.Q THEN
		_Error :=TRUE;
		strStatus:='Cylinder.List.fbUpCV_DiameterClamp M_Retract Timeout';
		END_IF
5800:
		Cylinder.List.fbUpCV_DiameterVert.M_Retract();
		 uiExecutingStep := 5900;
5900:
		tonDiameterTimeoutTwo.IN :=TRUE;
		IF Cylinder.List.fbUpCV_DiameterVert.InRearPosition THEN
			tonDiameterTimeoutTwo.IN :=FALSE;
		uiExecutingStep :=6000;
		END_IF
		IF tonDiameterTimeoutTwo.Q THEN
		_Error :=TRUE;
		strStatus:='Cylinder.List.fbUpCV_DiameterVert M_Retract Timeout';
		END_IF
6000:
		_Executed:= TRUE;





END_CASE
	
IF NOT Execute THEN
	eState:=STATE_RESETTING;
END_IF
IF _Error THEN
	eState:=STATE_ERROR;
END_IF
IF _Abort THEN
	eSTATE:=STATE_ABORTING;
END_IF
IF _Executed THEN
	eSTATE:=STATE_Done;
END_IF
END_METHOD

METHOD  M_STATE_RESETTING
VAR_INPUT
END_VAR
Error :=FALSE;
Done :=FALSE;
Busy := FALSE;


CASE uiResettingStep OF
	0 : 
		
		IF Cylinder.List.fbUpCV_DiameterHoriz.xError THEN
			Cylinder.List.fbUpCV_DiameterHoriz.M_Reset();
		END_IF
		IF Cylinder.List.fbUpCV_DiameterVert.xError THEN
			Cylinder.List.fbUpCV_DiameterVert.M_Reset();
		END_IF
		IF Cylinder.List.fbUpCV_DiameterClamp.xError THEN
			Cylinder.List.fbUpCV_DiameterClamp.M_Reset();
		END_IF
		uiResettingStep:=100;
		
	100:
		Cylinder.List.fbUpCV_DiameterVert.M_Retract();
		IF Cylinder.List.fbUpCV_DiameterClamp.InFrontPosition THEN
			uiResettingStep:=1000;
		ELSE
			uiResettingStep:=2000;	
		END_IF
	1000:
			
			IF Cylinder.List.fbUpCV_DiameterVert.InRearPosition THEN
				Cylinder.List.fbUpCV_DiameterHoriz.M_Extend();
				uiResettingStep:=1200;
			END_IF
	1200:		
			IF Cylinder.List.fbUpCV_DiameterHoriz.InFrontPosition THEN
				Cylinder.List.fbUpCV_DiameterClamp.M_Retract();
				uiResettingStep:=1300;
			END_IF
	1300:	
			IF Cylinder.List.fbUpCV_DiameterClamp.InRearPosition THEN
				uiResettingStep:=2000;
			END_IF
		
	2000 : 
			Cylinder.List.fbUpCV_DiameterHoriz.M_Retract();
				uiResettingStep:=2100;
	2100:
			IF Cylinder.List.fbUpCV_DiameterHoriz.InRearPosition THEN
				uiResettingStep:=9999;	
			END_IF
			
	9999:
		_ResetCompleted:=TRUE;
END_CASE
IF _ResetCompleted THEN
	eSTATE:=STATE_DORMANT;
END_IF
END_METHOD

END_FUNCTION_BLOCK

// ---- Library/20_MachineUnits/21_StorageArea/Service/FB_UpperFeedInConveyor.TcPOU
FUNCTION_BLOCK FB_UpperFeedInConveyor EXTENDS FB_ObjectBase_V2
VAR_INPUT
	
	_fbDiameterMovement : REFERENCE TO FB_DiameterMovement;
	
	Cylinder 	: REFERENCE TO UNI_CylinderList;
	Motor	 	: REFERENCE TO UNI_MotorList;
	Input 	 	: REFERENCE TO ST_InputTable;
	OutPut	 	: REFERENCE TO ST_OutputTable;
	
	Info		: ST_Auto_UpperFeedInConveyorInfo;
	
	AddingBox	: BOOL;
//    Execute    :BOOL;   // True : This prog will start.
//    Abort      :BOOL;   // True : This prog will be abort.
//    Reset      :BOOL;   // True : This prog will be reset.
//    ObjectName :STRING; // Set this fb name(About it's action)
END_VAR

VAR_OUTPUT
//	Status		: ST_StatusBasic;
	FeedBack    : ST_Auto_UpperFeedInConveyorFeedback;	
	_bForceUpperCV_Use	: BOOL;	
//    Busy    :BOOL;        // True : This prog is running.
//    Done    :BOOL;        // True : Command has been executed.
//    Aborted :BOOL;        // True : This prog is aborted.
//    Error   :BOOL;        // True : This prog has an error.
//    ErrorID :UINT;       // Output ErrorID
//    Status  :T_MaxString; // Output this prog status by string(255bytes)
END_VAR

VAR
//    eState :E_MethodStatus_Basic;
//	uiExecutingStep : UDINT; // This var is used to been controll STATE_EXECUTING process.
//	uiResettingStep : UDINT;
//	uiAbortingStep : UDINT;
//	_Executed :BOOL; // Executing process completed.
//	_Error : BOOL; // FB has an error.
//	_ResetCompleted : BOOL; // FB resetting completed.
//	_AbortCompleted : BOOL; // FB aborting completed.
	_Abort		: BOOL;
	strStatus	: T_MaxString;
	uiResumeStep : UINT;
	iMoveConveyor	:INT;// 1 = MoveForward , -1 = Move reverse , 0 or other = Stop
	tonUpperConveyorTimeOut			:TON;
	tonUpperConveyorDelay			:TON;
	tonUpperTimeOut					:TON;
	tonUpperTimeOutFive 			:TON;
	tonWaitSecondBoxArriveTimeout 	:TON;
	tonFeedAirBlowtime 				:TON;
	tonReverseConveyorDelay			:TON;
	TON_CheckHaveBox				:TON ;
	NoFirstBoxDiameter : BOOL;
	SecondBox	:BOOL;
	bSecondBoxInCameraPos :BOOL;
	uiFirstBoxDiameterStep :UINT :=0;
	uiSecondBoxAirBlowStep :UINT :=0;
	_UniqueErrorCode :STRING;
	
	
	//record time for C# photo
	tRecordTimer 		: ARRAY [1..100] OF TIME;
	tRecordFirstTimer	: ARRAY [1..100] OF TIME;
	tRecordSecondTimer	: ARRAY [1..100] OF TIME;
	TON_RecordTimer 	: TON;
	TON_RecordFirstTimer		: TON ;
	TON_RecordSecondTimer		: TON;
	TSaveTime					: TIME;
	TSaveFirstTime				: TIME;
	TSaveSecondTime				: TIME;
	iArrayNumber 				: INT :=1;
	iResetNumber				: INT;
	bResetRecordInfo			: BOOL;
	
	
END_VAR

A00_BasicUnits();
SUPER^.A10_StateControl();

ACTION A00_BasicUnits:
tonUpperConveyorTimeOut(PT:=T#20S);
tonUpperConveyorDelay();
tonUpperTimeOut(PT:=T#5.0S);
tonUpperTimeOutfive(PT:=T#60S);
tonWaitSecondBoxArriveTimeout(PT:=T#20S);
tonFeedAirBlowtime(PT:=info.FeedAirblowTime);
tonReverseConveyorDelay(PT:=T#6S);
TON_CheckHaveBox(PT :=T#35S);
ErrorID :=2710;



TON_RecordTimer (PT:=T#1D);
TON_RecordFirstTimer (PT := T#1D);
TON_RecordSecondTimer (PT := T#1D);

// only for record the photo time use
IF bResetRecordInfo THEN
	FOR iResetNumber :=1 TO 100 DO
		tRecordTimer[iResetNumber] :=T#0S;
		tRecordFirstTimer[iResetNumber] :=T#0S;
		tRecordSecondTimer[iResetNumber] :=T#0S;
	END_FOR
END_IF
END_ACTION

METHOD GetModelState
VAR_OUTPUT
    xDone    :BOOL;
    xBusy    :BOOL;
    xError   :BOOL;
    xAborted :BOOL;
    iErrorID :UDINT;
	UniqueErrorCode : STRING;
END_VAR
xDone    := Done;
xBusy    := Busy;
xError   := Error;
xAborted := Abort;
iErrorID := ErrorID;
END_METHOD

METHOD GetName : STRING
GetName := ObjectName;
END_METHOD

METHOD  M_STATE_ABORTED
VAR_INPUT
END_VAR
ERROR :=TRUE;
Busy := FALSE;
Aborted := TRUE;
_Abort := FALSE;
UniqueErrorCode:=_UniqueErrorCode;
SUPER^.Status := strStatus;

IF NOT Execute THEN
	eSTATE:=STATE_RESETTING;
	
ELSIF Execute AND Reset THEN

		CASE uiExecutingStep OF
			20:
				uiExecutingStep :=10;
				strStatus :='prepare cylinders retry';
				
			100:
				uiExecutingStep :=100;
				strStatus :='check no box retry';
			200:
				uiExecutingStep :=200;
				strStatus :='check Block3Cylinder retry';

			400://將讀碼壓盒1 往後 重做一次
				Cylinder.List.fbUpCV_CamaraPress1.M_Retract();
				IF Cylinder.List.fbUpCV_CamaraPress1.InRearPosition THEN
				uiExecutingStep :=300;
				strStatus :='check ReadCodeBox1 infrontposition retry';
				END_IF
			460:	//Box1 done step abort
				uiExecutingStep :=450;
				strStatus :='Check FirstBoxCamaraDone info retry';
			550:
				uiExecutingStep :=500;
				strStatus :='ReadCodePressBox1Cylinder and FeedInBlockBox3Cylinder Backward retry';
			600:
				uiExecutingStep :=600;
				strStatus :='FirstBoxCameraDiameterRequest Info retry';
			610:
				uiExecutingStep :=610;
				strStatus :='CodeReadingBoxDetection first box leave retry';
			700:
				uiExecutingStep :=700;
				strStatus :='UpperFeedInBlockBox2Cylinder MoveForward retry';
			800:
				uiExecutingStep :=800;
				strStatus :='Box not at UpperBox2Detection retry ';
				
			1000:
				Cylinder.List.fbUpCV_DiameterPress.M_Retract();
				IF Cylinder.List.fbUpCV_DiameterPress.InRearPosition THEN
					uiExecutingStep :=800;
					strStatus :='DiameterMeasurementPressBoxCylinder MoveBackward retry';
				END_IF
			1200:
				Cylinder.List.fbUpCV_CamaraPress1.M_Retract();
				Cylinder.List.fbUpCV_CamaraPress2.M_Retract();
				IF Cylinder.List.fbUpCV_CamaraPress1.InRearPosition AND 
					Cylinder.List.fbUpCV_CamaraPress2.InRearPosition THEN
					uiExecutingStep :=1100;
					strStatus :='ReadCodePressBox 1 and 2 Cylinder retry';
				END_IF
			1300:
				uiExecutingStep :=1300;
				strStatus :='SecondBoxCameraDone info retry';
			1400:
				uiExecutingStep :=1400;
				strStatus :='FirstBoxCameraDiameterDone info retry';
			1600:
				uiExecutingStep :=1500;
				strStatus :='DiameterMeasurementPressBoxCylinder and FeedInBlockBox2Cylinder MoveBackward retry';
			1700:
				uiExecutingStep :=1700;
				strStatus :='check UpperBox2Detection have box';
			1800:
				Cylinder.List.fbUpCV_DiameterPress.M_Retract();
				IF Cylinder.List.fbUpCV_DiameterPress.InRearPosition THEN
				uiExecutingStep :=1700;
				strStatus :='DiameterMeasurementPressBoxCylinder Forward retry';
				END_IF
			1900:
				uiExecutingStep :=1900;
				strStatus :='DiameterMovement PickDone  retry';
			2000:
				uiExecutingStep :=2000;
				strStatus :='SecondBoxCameraDiameterDone retry';
			2100:	
				uiExecutingStep :=2100;
				strStatus :='_fbDiameterMovement done retry';
			2200:
				
				
		END_CASE
	
	eSTATE:=STATE_EXECUTING;
	
END_IF
END_METHOD

METHOD  M_STATE_ABORTING
VAR_INPUT
END_VAR
Busy :=FALSE;
CASE uiAbortingStep OF
	0:
		tonUpperConveyorTimeOut.IN 	:=FALSE;
		tonUpperConveyorDelay.IN	:=FALSE;
		tonUpperTimeOut.IN 			:=FALSE;
		tonUpperTimeOutfive.IN		:=FALSE;
		TON_CheckHaveBox.IN 		:=FALSE;
		uiAbortingStep :=100;
	100:
		Motor.List.UpCV.M_MotorStop();
		OutPut.bCamara_Blow :=FALSE;
		IF Motor.List.UpCV.InStopped THEN
			uiAbortingStep :=9999;
		END_IF
	9999:	
		_AbortCompleted:=TRUE;
END_CASE

IF _AbortCompleted THEN	
	eSTATE :=STATE_ABORTED;
END_IF
END_METHOD

METHOD  M_STATE_DONE
VAR_INPUT
END_VAR
Busy := FALSE;
Done:=TRUE;
_fbDiameterMovement.Execute := FALSE;
_fbDiameterMovement.bContinue:=FALSE;
IF NOT Execute THEN
	eSTATE:=STATE_RESETTING;
END_IF
END_METHOD

METHOD  M_STATE_DORMANT
VAR_INPUT
END_VAR
Busy    := FALSE;
Done    := FALSE;
Aborted := FALSE;
Error   := FALSE;
FeedBack.InterventionRequest :=FALSE;
strStatus :='No Error';
uiExecutingStep :=0;
uiResettingStep	:=0;
NoFirstBoxDiameter:= SecondBox:=FALSE;
tonUpperConveyorTimeOut.IN := FALSE;
tonUpperConveyorDelay.IN :=FALSE;
tonUpperTimeOut.IN :=FALSE;
tonUpperTimeOutFive.IN :=FALSE;
tonWaitSecondBoxArriveTimeout.IN :=FALSE;
TON_CheckHaveBox.IN :=false;
tonFeedAirBlowtime.IN :=false;
bSecondBoxInCameraPos := FALSE;
_bForceUpperCV_Use := false;
_Abort := _Executed := _Error:= _ResetCompleted:=_AbortCompleted:=FALSE;
iMoveConveyor := 0;
uiFirstBoxDiameterStep  :=0;
uiSecondBoxAirBlowStep	:=0;
_UniqueErrorCode :='0';
IF Execute THEN
	eSTATE:=STATE_EXECUTING;
END_IF
END_METHOD

METHOD  M_STATE_ERROR
VAR_INPUT
END_VAR
ERROR :=TRUE;
Busy :=FALSE;
UniqueErrorCode:=_UniqueErrorCode;
SUPER^.Status := strStatus;
_fbDiameterMovement.Execute := FALSE;


Motor.List.UpCV.M_MotorStop(); 
OutPut.bCamara_Blow :=FALSE;

IF NOT Execute THEN	
eSTATE:=STATE_RESETTING;
END_IF
END_METHOD

METHOD  M_STATE_EXECUTING
VAR_INPUT
END_VAR

VAR_INST
	
	
END_VAR
VAR
	END_I: INT;
	
END_VAR
Busy :=TRUE;

//Conveyor motor control
CASE iMoveConveyor OF
	1:
	Motor.list.UpCV.M_MoveForward();
	Cylinder.List.fbUpCV_CamaraPress4.M_Retract(); //Feedin working , open the end to allow box feedin
	//OutPut.bCamara_Blow :=TRUE;
	-1:
	Motor.list.UpCV.M_MoveBackward();
	Cylinder.List.fbUpCV_CamaraPress4.M_Retract(); //Feedin working , open the end to allow box feedin
ELSE		
	Motor.list.UpCV.M_MotorStop();
	Cylinder.List.fbUpCV_CamaraPress4.M_Extend();// End feedin , block the conveyor in case no one push boxes in working area
	//OutPut.bCamara_Blow :=FALSE;		change use airflow to take photo before
END_CASE



CASE uiExecutingStep OF
	
0 : // StandBy
	TON_RecordTimer.IN := TRUE;
	iMoveConveyor:=0;
	tonUpperConveyorTimeOut.IN:=FALSE;
	tonUpperConveyorDelay.IN :=FALSE;
	tonUpperConveyorDelay.PT:=T#200MS;
	IF Info.NrOfBox=1 THEN
		SecondBox:=FALSE;
	ELSIF Info.NrOfBox=2 THEN
		SecondBox:=TRUE;	
	ELSE
	_Error := TRUE;
	  strStatus := 'Data not correct';		
	END_IF
	uiExecutingStep :=10;

10: //Prepare cylinders
	IF Cylinder.List.fbUpCV_FeedInPress1.xError THEN
		Cylinder.List.fbUpCV_FeedInPress1.M_Reset();
	END_IF
	IF Cylinder.List.fbUpCV_FeedInPress2.xError THEN
		Cylinder.List.fbUpCV_FeedInPress1.M_Reset();
	END_IF
	IF Cylinder.List.fbUpCV_DiameterPress.xError THEN
		Cylinder.List.fbUpCV_DiameterPress.M_Reset();
	END_IF
	IF Cylinder.List.fbUpCV_CamaraPress1.xError THEN
		Cylinder.List.fbUpCV_CamaraPress1.M_Reset();
	END_IF
	IF Cylinder.List.fbUpCV_CamaraPress2.xError THEN
		Cylinder.List.fbUpCV_CamaraPress2.M_Reset();
	END_IF
	IF Cylinder.List.fbUpCV_CamaraPress4.xError THEN
		Cylinder.List.fbUpCV_CamaraPress4.M_Reset();
	END_IF
	IF Cylinder.List.fbUpCV_Block1.xError THEN
		Cylinder.List.fbUpCV_Block1.M_Reset();
	END_IF
	IF Cylinder.List.fbUpCV_Block2.xError THEN
		Cylinder.List.fbUpCV_Block2.M_Reset();
	END_IF
	IF Cylinder.List.fbUpCV_Block3.xError THEN
		Cylinder.List.fbUpCV_Block3.M_Reset();
	END_IF
	IF Motor.List.UpCV.xError THEN
		Motor.List.UpCV.M_Reset();
	END_IF
	
	uiExecutingStep :=20;
	
20: //Prepare cylinders
	tonUpperTimeOut.IN :=TRUE;
	Cylinder.List.fbUpCV_FeedInPress1.M_Retract();		(* Cylinder.List.fbUpCV_FeedInPress1.M_Retract();*)	
	Cylinder.List.fbUpCV_FeedInPress2.M_Retract();		(*Cylinder.List.fbUpCV_FeedInPress2.M_Retract();*)
	Cylinder.List.fbUpCV_DiameterPress.M_Retract();		(*Cylinder.List.fbUpCV_DiameterPress.M_Retract();*)
	Cylinder.List.fbUpCV_CamaraPress1.M_Retract();		(*Cylinder.List.fbUpCV_CamaraPress1.M_Retract();*)		
	//Cylinder.List.fbUpCV_CamaraPress2.M_Retract();	(*Cylinder.List.fbUpCV_CamaraPress2.M_Retract();*)
	Cylinder.List.fbUpCV_CamaraPress4.M_Retract();		(*Cylinder.List.fbUpCV_CamaraPress4.M_Retract();*)	
	Cylinder.List.fbUpCV_Block1.M_Retract();			(*Cylinder.List.fbUpCV_Block1.M_Retract();*)
	Cylinder.List.fbUpCV_Block2.M_Retract();			(*Cylinder.List.fbUpCV_Block2.M_Retract();*)
	Cylinder.List.fbUpCV_Block3.M_Retract();			(*Cylinder.List.fbUpCV_Block3.M_Retract();*)

	//edit by Min 20250326
	IF Cylinder.List.fbUpCV_FeedInPress1.InRearPosition AND		
		Cylinder.List.fbUpCV_FeedInPress2.InRearPosition AND
		Cylinder.List.fbUpCV_DiameterPress.InRearPosition AND
		Cylinder.List.fbUpCV_CamaraPress1.InRearPosition AND
		Cylinder.List.fbUpCV_CamaraPress4.InRearPosition AND
		Cylinder.List.fbUpCV_Block1.InRearPosition AND
		Cylinder.List.fbUpCV_Block2.InRearPosition AND
		Cylinder.List.fbUpCV_Block3.InRearPosition THEN
		
		tonUpperTimeOut.IN :=FALSE;
		uiExecutingStep :=100;	
	END_IF
	IF tonUpperTimeOut.Q THEN
		_Abort :=TRUE;
		strStatus :='Prepare Cylinder clear command timeout';
	END_IF
	
100:// Check No Box 
	IF Input.bUpCV_Block1Detect_Sensor OR 
	  Input.bUpCV_Block2Detect_Sensor OR
	  Input.bUpCV_BoxArrived_Sensor OR
	  Input.bUpCV_Block3Detect_Sensor THEN
	 	 IF NOT AddingBox THEN
		 _bForceUpperCV_Use := TRUE;		//force UpperCV for Backward CV use
	 	 uiExecutingStep :=110; //Try reverse conveyor 
			ELSE 
			  _Abort := TRUE;
		 	 strStatus := 'Conveyor not ready , please remove boxes in front';
		  END_IF
	 ELSE
 		uiExecutingStep :=200; 
	 END_IF
110:
		iMoveConveyor:= -1;
		Cylinder.List.fbUpCV_CamaraPress2.M_Retract();
		tonReverseConveyorDelay.IN :=TRUE;
		uiExecutingStep :=120;

120:
		//tonFeedAirBlowtime.IN :=TRUE;
		IF tonReverseConveyorDelay.Q THEN
			iMoveConveyor :=0;
			uiExecutingStep :=130; 
		END_IF
130:
		tonReverseConveyorDelay.IN :=FALSE;
		IF Input.bUpCV_Block1Detect_Sensor OR 
		  Input.bUpCV_Block2Detect_Sensor OR
		  Input.bUpCV_BoxArrived_Sensor OR
	 	 Input.bUpCV_Block3Detect_Sensor THEN 
			  _Abort := TRUE;
		 	 strStatus := 'Conveyor not ready , please remove boxes in front';
		 ELSE
			uiExecutingStep :=140; 	 
		 END_IF		
140:
   		IF Motor.list.UpCV.InStopped THEN
			uiExecutingStep :=200;
		END_IF
200: // motor start and camera block up 
	_bForceUpperCV_Use := FALSE;		//release UpperCV force use 
	tonUpperConveyorTimeOut.IN:=TRUE;
	iMoveConveyor:=1;
	Cylinder.List.fbUpCV_CamaraPress2.M_Retract();
	Cylinder.List.fbUpCV_Block3.M_Extend();
	IF Cylinder.List.fbUpCV_Block3.InFrontPosition AND
		Cylinder.List.fbUpCV_CamaraPress2.InRearPosition THEN
		tonUpperConveyorTimeOut.IN:=FALSE;
		uiExecutingStep :=300;
	END_IF
	IF tonUpperConveyorTimeOut.Q THEN
	  _Error := TRUE;
	  strStatus := 'Cylinder.List.fbUpCV_Block3 timeout';
	END_IF
		  
	  
300://Dtect camera sensor and wait first box arrive in camera position
	TON_CheckHaveBox.IN :=TRUE;
	tonUpperConveyorDelay.IN:=Input.bUpCV_Block3Detect_Sensor; //Delay a moment to make sure box move till end of block 	
	IF tonUpperConveyorDelay.Q THEN
			TON_CheckHaveBox.IN :=FALSE;
			Cylinder.List.fbUpCV_CamaraPress1.M_Extend(); //Press box 
			tonUpperConveyorDelay.IN := FALSE;
			uiExecutingStep :=400;			
	END_IF
	IF TON_CheckHaveBox.Q THEN	//if behind not have box feedback box = 0
		uiExecutingStep := 2700;
	END_IF
	
400:// Check pressing job done for first box in camera position	
	tonUpperTimeOut.IN :=TRUE;
	IF Cylinder.List.fbUpCV_CamaraPress1.InFrontPosition THEN
		tonUpperTimeOut.IN := FALSE;
		Cylinder.List.fbUpCV_CamaraPress2.M_Extend();
		uiExecutingStep :=450;		
	END_IF
	IF tonUpperTimeOut.Q THEN
		_Abort := TRUE;
		strStatus := 'Cylinder.List.fbUpCV_CamaraPress1.M_MoveForward timeout';
	END_IF

450:// send first box camera signal
	
	tonFeedAirBlowtime.IN :=TRUE;
	OutPut.bCamara_Blow :=TRUE;
	IF tonFeedAirBlowtime.Q THEN
		tonFeedAirBlowtime.IN:=FALSE;
		OutPut.bCamara_Blow :=FALSE;
		FeedBack.FirstBoxCamera :=TRUE;
		TON_RecordFirstTimer.IN :=TRUE;
		uiExecutingStep :=460;
	END_IF
	

460: // Wait first box camera done
	// todo : timeout
	tonUpperTimeOutFive.IN :=TRUE;		//T#5S
	IF Info.FirstBoxCameraDone THEN
		tonUpperTimeOutFive.IN :=FALSE;
		FeedBack.FirstBoxCamera :=FALSE;
		uiExecutingStep :=500;
	END_IF	
	IF tonUpperTimeOutFive.Q THEN
		_Abort :=TRUE;
		strStatus := 'C# FirstBoxCameraDone timeout';
	END_IF
	
500://Let first box move forward
	TSaveFirstTime 	:= TON_RecordFirstTimer.ET;
	TON_RecordFirstTimer .IN :=FALSE;
	Cylinder.List.fbUpCV_CamaraPress1.M_Retract(); // release press
	Cylinder.List.fbUpCV_Block3.M_Retract();//release blocker todo : add description
	uiExecutingStep :=550;
	
550://check cylinder inrearposition		edit by Min 20250326
	tonUpperTimeOut.IN :=TRUE;
	IF Cylinder.List.fbUpCV_CamaraPress1.InRearPosition AND		
		Cylinder.List.fbUpCV_Block3.InRearPosition THEN
		
		uiExecutingStep :=600;
	END_IF
	IF tonUpperTimeOut.Q THEN
		_Abort := TRUE;
		strStatus := 'Cylinder.List.fbUpCV_CamaraPress1 or Cylinder.List.fbUpCV_Block3 InRearPosition timeout';
	END_IF
	
600://Check if diameter camera needed
	tonUpperTimeOut.IN :=FALSE;
	tonUpperTimeOutFive.IN :=TRUE;
	IF Info.FirstBoxCameraDiameterRequest THEN
		tonUpperTimeOutFive.IN :=FALSE;
		uiExecutingStep :=700;
		ELSE
			IF SecondBox THEN
				tonUpperTimeOutFive.IN :=FALSE;
				NoFirstBoxDiameter:=TRUE;
				uiExecutingStep :=610;//Only if box 1 no need to measure diameter
			ELSE
				tonUpperTimeOutFive.IN :=FALSE;
				uiExecutingStep :=2400;	
			END_IF
	END_IF
	IF tonUpperTimeOutFive.Q THEN
		_Abort := TRUE;
		strStatus :='C# FirstBoxCameraDiameterRequest timeout';
	END_IF
	
610: //Check Box 1 leave read code camera position
	tonUpperTimeOut.IN :=TRUE;
	tonUpperConveyorDelay.IN := NOT Input.bUpCV_Block3Detect_Sensor;
	IF tonUpperConveyorDelay.Q THEN
		tonUpperConveyorDelay.IN :=FALSE;
		uiExecutingStep :=620;
	END_IF
	IF tonUpperTimeOut.Q  THEN
		_Abort :=TRUE;
		strStatus :='Input.bUpCV_Block3Detect_Sensor first box leave timeout';
	END_IF
	
620: // Leave Box 2				//timeout and Check InRearPositonEdit by Min 20250326	
		tonUpperTimeOut.IN :=FALSE;	
		IF SecondBox THEN			
			Cylinder.List.fbUpCV_CamaraPress2.M_Retract(); //Release press box
			Cylinder.List.fbUpCV_Block3.M_Extend(); //release blocker
			IF Cylinder.List.fbUpCV_CamaraPress2.InRearPosition AND Cylinder.List.fbUpCV_Block3.InFrontPosition THEN
				uiExecutingStep :=1100;
			END_IF
		END_IF
		
700: //Rise diameter blocker
	tonUpperTimeOut.IN :=TRUE;
	Cylinder.List.fbUpCV_Block2.M_Extend();
	IF Cylinder.List.fbUpCV_Block2.InFrontPosition THEN
		tonUpperTimeOut.IN :=FALSE;
		uiExecutingStep :=800;
	END_IF
	IF tonUpperTimeOut.Q THEN
		_Abort :=TRUE;
		strStatus :='Cylinder.List.fbUpCV_Block2 MoveForward timeout';
	END_IF
800: // wait first box ready on diameter position
	tonUpperTimeOut.IN :=TRUE;
	tonUpperConveyorDelay.IN:=Input.bUpCV_Block2Detect_Sensor;
	IF tonUpperConveyorDelay.Q THEN
		tonUpperTimeOut.IN :=FALSE;
		tonUpperConveyorDelay.IN:=FALSE;
		Cylinder.List.fbUpCV_DiameterPress.M_Extend();
		
		IF SecondBox THEN	
			tonUpperTimeOut.IN :=FALSE;		
			Cylinder.List.fbUpCV_CamaraPress2.M_Retract();
			Cylinder.List.fbUpCV_Block3.M_Extend();
		END_IF
		uiExecutingStep :=1000;
	END_IF
	IF tonUpperTimeOut.Q THEN
		_Abort :=TRUE;
		strStatus :='Box not at Input.bUpCV_Block2Detect_Sensor ';
	END_IF
	
1000: // Wait diameter blocker ready
	tonUpperTimeOut.IN :=TRUE;
	IF 	Cylinder.List.fbUpCV_DiameterPress.InFrontPosition THEN
		tonUpperTimeOut.IN :=FALSE;
		uiExecutingStep :=1100;
	END_IF
	IF tonUpperTimeOut.Q THEN
		_Abort :=TRUE;
		strStatus :='Cylinder.List.fbUpCV_DiameterPress MoveForward timeout';
	END_IF

1100: // Pick needle to diameter camera

		
		CASE uiFirstBoxDiameterStep OF
			
		0:
			IF NOT NoFirstBoxDiameter THEN
	  			_fbDiameterMovement.Execute := TRUE;
				uiFirstBoxDiameterStep:=100;
			ELSE
				uiFirstBoxDiameterStep:=9000;	
	  		END_IF
		
		100:
			IF _fbDiameterMovement.Busy THEN
				uiFirstBoxDiameterStep:=200;
			END_IF	
			
		200:
			tonUpperTimeOutFive.IN :=TRUE;
			 IF _fbDiameterMovement.PickDone THEN
				  tonUpperTimeOutFive.IN :=FALSE;
				  FeedBack.FirstBoxCameraDiameter:=TRUE;		  
			  END_IF
			 IF Info.FirstBoxCameraDiameterDone THEN
				tonUpperTimeOutFive.IN:=FALSE;
				 FeedBack.FirstBoxCameraDiameter:=FALSE;
			 	_fbDiameterMovement.bContinue:=TRUE;
			 	uiFirstBoxDiameterStep:=300;
			  END_IF
			 IF tonUpperTimeOutFive.Q THEN
				 _Error :=TRUE;
				 strStatus :='box1 diameter timeout';
			 END_IF
		300:
			 IF _fbDiameterMovement.Done THEN
				  uiFirstBoxDiameterStep:=9000;		  
			  END_IF	  
		
		9000:
				_fbDiameterMovement.bContinue:=FALSE;
				_fbDiameterMovement.Execute:=FALSE;
				Cylinder.List.fbUpCV_DiameterPress.M_Retract();
				Cylinder.List.fbUpCV_Block2.M_Retract();
				// first box leave	  
				
				IF bSecondBoxInCameraPos AND 
					Cylinder.List.fbUpCV_DiameterPress.InRearPosition AND
					Cylinder.List.fbUpCV_Block2.InRearPosition THEN
					
					uiExecutingStep :=1200;
				END_IF
		END_CASE
						
		
	  		IF SecondBox THEN
				tonWaitSecondBoxArriveTimeout.IN :=TRUE;
	  			tonUpperConveyorDelay.IN := Input.bUpCV_Block3Detect_Sensor;
 				IF tonUpperConveyorDelay.Q THEN								
					tonUpperConveyorDelay.IN:=FALSE;
					tonWaitSecondBoxArriveTimeout.IN :=FALSE;
					Cylinder.List.fbUpCV_CamaraPress2.M_Extend();
					Cylinder.List.fbUpCV_CamaraPress1.M_Extend();
//					bSecondBoxInCameraPos :=TRUE;
				END_IF	
	 		 ELSE
				 bSecondBoxInCameraPos:=TRUE;
	 		 END_IF
			 
		CASE uiSecondBoxAirBlowStep OF
			 0:
			 	IF 	Cylinder.List.fbUpCV_CamaraPress1.InFrontPosition AND 
					Cylinder.List.fbUpCV_CamaraPress2.InFrontPosition THEN
						uiSecondBoxAirBlowStep :=10;
				END_IF
			10:
				OutPut.bCamara_Blow :=TRUE;		//take photo need airflow before
				tonFeedAirBlowtime.IN :=TRUE;
					IF tonFeedAirBlowtime.Q THEN		
						tonFeedAirBlowtime.IN :=FALSE;
						OutPut.bCamara_Blow :=FALSE;
						FeedBack.SecondBoxCamera:=TRUE;
						TON_RecordSecondTimer.IN :=TRUE;
						uiSecondBoxAirBlowStep :=20;
					END_IF
			20:
				IF Info.SecondBoxCameraDone THEN
					uiSecondBoxAirBlowStep :=30;
					TSaveSecondTime := TON_RecordSecondTimer.ET;
				END_IF
			30:	
					
					
					TON_RecordSecondTimer.IN :=FALSE;
					bSecondBoxInCameraPos:=TRUE;	
			
		END_CASE
		
//			IF Cylinder.List.fbUpCV_CamaraPress1.InFrontPosition AND 
//				Cylinder.List.fbUpCV_CamaraPress2.InFrontPosition THEN
//				OutPut.bCamara_Blow :=TRUE;		//take photo need airflow before
//				tonFeedAirBlowtime.IN :=TRUE;
//					IF tonFeedAirBlowtime.Q THEN		
//						tonFeedAirBlowtime.IN :=FALSE;
//						OutPut.bCamara_Blow :=FALSE;
//						FeedBack.SecondBoxCamera:=TRUE;	
//							IF Info.SecondBoxCameraDone THEN
//								bSecondBoxInCameraPos:=TRUE;	
//							END_IF	
//					END_IF
//			END_IF
	  
	  IF tonUpperConveyorTimeOut.Q THEN
			_Error :=TRUE;
			strStatus:='First box diameter timeout';		
		  
	  END_IF
		IF tonWaitSecondBoxArriveTimeout.Q THEN
			IF Input.bUpCV_ReLoadDetect_Sensor THEN
				_Error :=TRUE;
				strStatus:='Second box feedin to read code camera pos timeout';		
			ELSE
				tonUpperConveyorTimeOut.IN :=FALSE;
				SecondBox :=FALSE;
			END_IF	 
		END_IF

1200: 	// If first box leave diameter sensor , let second box go
		tonUpperTimeOut.IN :=TRUE;
		tonUpperConveyorDelay.PT:=T#600MS;		
		tonUpperConveyorDelay.IN := NOT Input.bUpCV_Block2Detect_Sensor;
		
		IF tonUpperConveyorDelay.Q THEN
			tonUpperConveyorDelay.IN :=FALSE;
			tonUpperTimeOut.IN :=FALSE;
			IF SecondBox AND INfo.SecondBoxCameraDiameterRequest THEN
				tonUpperTimeOut.IN :=FALSE;
				Cylinder.List.fbUpCV_Block2.M_Extend();
				Cylinder.List.fbUpCV_CamaraPress1.M_Retract();
				Cylinder.List.fbUpCV_Block3.M_Retract();
				uiExecutingStep :=1700;
			ELSE
				tonUpperTimeOut.IN :=FALSE;
				uiExecutingStep :=2400;	
			END_IF

		END_IF
		IF tonUpperTimeOut.Q THEN
			_Abort :=TRUE;
			strStatus :='First box still at Input.bUpCV_Block2Detect_Sensor';
		END_IF

1700: //Second box diameter request
		tonUpperTimeOut.IN :=TRUE;
		tonUpperConveyorDelay.IN :=Input.bUpCV_Block2Detect_Sensor;
		IF tonUpperConveyorDelay.Q THEN
			tonUpperTimeOut.IN :=FALSE;
			tonUpperConveyorDelay.IN :=FALSE;
			Cylinder.List.fbUpCV_DiameterPress.M_Extend();
			uiExecutingStep :=1800;
		END_IF
		IF tonUpperTimeOut.Q THEN
			_Abort :=TRUE;
			strStatus :='Input.bUpCV_Block2Detect_Sensor not have box';
		END_IF
1800: //wait second box in diameter position
		tonUpperTimeOut.IN :=TRUE;
		IF Cylinder.List.fbUpCV_DiameterPress.InFrontPosition THEN
			tonUpperTimeOut.IN :=FALSE;
			uiExecutingStep :=1900;
		END_IF
		IF tonUpperTimeOut.Q THEN
			_Abort :=TRUE;
			strStatus :='Cylinder.List.fbUpCV_DiameterPress MoveForward timeout';
			
		END_IF
		
